text list "SINAMICS_G120_FW4.4_faults": 0 'No fault / Keine Störung'; 1000 'Internal software error / Softwarefehler intern'; 1001 'FloatingPoint exception / FloatingPoint Ausnahme'; 1002 'Internal software error / Softwarefehler intern'; 1003 'Acknowledgement delay when accessing the memory / Quittungsverzug bei Speicherzugriff'; 1004 'Internal software error / Softwarefehler intern'; 1005 'File upload/download error / Datei Upload/Download fehlgeschlagen'; 1009 'CU: Control module overtemperature / CU: Regelungsbaugruppe Übertemperatur'; 1010 'Drive type unknown / Antriebstyp unbekannt'; 1011 'Download interrupted / Download abgebrochen'; 1012 'Project conversion error / Projekt Konvertierungsfehler'; 1013 'CU: Fan operating time reached or exceeded / CU: Betriebsdauer Lüfter erreicht oder überschritten'; 1015 'Internal software error / Softwarefehler intern'; 1016 'Firmware changed / Firmware verändert'; 1017 'Component lists changed / Komponentenlisten verändert'; 1018 'Booting has been interrupted several times / Hochlauf mehrmals abgebrochen'; 1019 'Writing to the removable data medium unsuccessful / Wechselmedium schreiben fehlgeschlagen'; 1020 'Write to RAM disk unsuccessful / RAM disk schreiben fehlgeschlagen'; 1023 'Software timeout (internal) / Software Timeout intern'; 1028 'Configuration error / Konfigurationsfehler'; 1030 'Sign-of-life failure for master control / Lebenszeichenausfall bei Steuerungshoheit'; 1031 'Sign-of-life failure for OFF in REMOTE / Lebenszeichenausfall bei AUS in REMOTE'; 1033 'Units changeover: Reference parameter value invalid / Einheitenumschaltung: Bezugsparameterwert ungültig'; 1034 'Units changeover: Calculation parameter values after reference value change unsuccessful Einheitenumschaltung: Berechnung Parameterwerte nach Bezugswertänderung fehlgeschlagen'; 1035 'ACX: Boot from the back-up parameter back-up files / ACX: Hochlauf erfolgt aus Backup-Parametersicherungsdateien'; 1036 'ACX: Parameter back-up file missing / ACX: Parametersicherungsdatei fehlt'; 1037 'ACX: Re-naming the parameter back-up file unsuccessful / ACX: Parametersicherungsdatei umbenennen fehlgeschlagen'; 1038 'ACX: Loading the parameter back-up file unsuccessful / ACX: Parametersicherungsdatei laden fehlgeschlagen'; 1039 'ACX: Writing to the parameter back-up file was unsuccessful / ACX: Parametersicherungsdatei schreiben fehlgeschlagen'; 1040 'Save parameter settings and carry out a POWER ON / Parameter sichern und POWER ON erforderlich'; 1041 'Parameter save necessary / Parameter sichern erforderlich'; 1042 'Parameter error during project download / Parameterfehler beim Projekt-Download'; 1043 'Fatal error at project download / Schwerer Fehler beim Projekt-Download'; 1044 'CU: Descriptive data error / CU: Beschreibungsdaten fehlerhaft'; 1045 'CU: Configuring data invalid / CU: Projektierungsdaten ungültig'; 1049 'It is not possible to write to file / Schreiben in Datei nicht möglich'; 1050 'Memory card and device incompatible / Speicherkarte und Gerät inkompatibel'; 1053 'CU: System overload measured / CU: Systemüberlastung gemessen'; 1054 'CU: System limit exceeded / CU: Systemgrenze überschritten'; 1064 'CU: Internal error (CRC) / CU: Interner Fehler (CRC)'; 1066 'Buffer memory: 70% fill level reached or exceeded / Zwischenspeicher: Füllstand 70 % erreicht oder überschritten'; 1067 'Buffer memory: 100 % fill level reached / Zwischenspeicher: Füllstand 100 % erreicht'; 1068 'CU: Data memory, memory overflow / CU: Datenspeicher Speicherüberlauf'; 1069 'Parameter backup and device incompatible / Parametersicherung und Gerät inkompatibel'; 1098 'RTC: Date and time setting required / RTC: Datum und Zeit einstellen erforderlich'; 1099 'Tolerance window of time synchronization exited / Toleranzfenster der Uhrzeitsynchronisation verlassen'; 1100 'CU: Memory card withdrawn / CU: Speicherkarte gezogen'; 1104 'CU: Do not power down. File system being optimized. / CU: Nicht ausschalten Optimierung Dateisystem läuft'; 1105 'CU: Insufficient memory / CU: Speicher nicht ausreichend'; 1107 'CU: Data save in the non-volatile memory unsuccessful / CU: Speichern in nichtflüchtigen Speicher fehlgeschlagen'; 1110 'CU: More than one SINAMICS G on one Control Unit / CU: Mehr als ein SINAMICS G an einer Control Unit'; 1111 'CU: Mixed operation of drive units illegal / CU: Mischbetrieb von Antriebsgeräten unzulässig'; 1112 'CU: Power unit not permissible / CU: Leistungsteil unzulässig'; 1120 'Terminal initialization has failed / Initialisierung Klemmen fehlgeschlagen'; 1122 'Frequency at the measuring probe input too high / Frequenz am Messtastereingang zu hoch'; 1150 'CU: Number of instances of a drive object type exceeded / CU: Anzahl Instanzen eines Antriebsobjekttyps überschritten'; 1151 'CU: Number of drive objects of a category exceeded / CU: Anzahl Antriebsobjekte einer Kategorie überschritten'; 1200 'CU: Time slice management internal software error / CU: Zeitscheibenmanagement Softwarefehler intern'; 1205 'CU: Time slice overflow / CU: Zeitscheibenüberlauf'; 1221 'CU: Bas clk cyc too low / CU: Basistakt zu klein'; 1223 'CU: Sampling time inconsistent / CU: Abtastzeit inkonsistent'; 1224 'CU: Pulse frequency inconsistent / CU: Pulsfrequenz inkonsistent'; 1250 'CU: CU-EEPROM incorrect read-only data / CU: CU-EEPROM Read-Only-Daten fehlerhaft'; 1251 'CU: CU-EEPROM incorrect read-write data / CU: CU-EEPROM Read-Write-Daten fehlerhaft'; 1255 'CU: Option Board EEPROM read-only data error / CU: Option Board EEPROM Read-Only-Daten fehlerhaft'; 1256 'CU: Option Board EEPROM read-write data error / CU: Option Board EEPROM Read-Write-Daten fehlerhaft'; 1275 'Hardware description error / Hardware-Beschreibung fehlerhaft'; 1276 'Hardware description not fully compatible / Hardware-Beschreibung nicht voll kompatibel'; 1303 'Function not supported / Funktion nicht unterstützt'; 1305 'Topology: Component number missing / Topologie: Komponentennummer fehlt'; 1314 'Topology: Component must not be present / Topologie: Komponente darf nicht vorhanden sein'; 1315 'Drive object not ready for operation / Antriebsobjekt nicht betriebsfähig'; 1316 'Drive object inactive and again ready for operation / Antriebsobjekt inaktiv und wieder betriebsfähig'; 1317 'De-activated component again present / Deaktivierte Komponente wieder vorhanden'; 1318 'BICO: De-activated interconnections present / BICO: Aufgelöste Verschaltungen vorhanden'; 1319 'Inserted component not initialized / Zugesteckte Komponente nicht initialisiert'; 1320 'Topology: Drive object number does not exist in configuration / Topologie: Antriebsobjektnummer fehlt in Konfiguration'; 1321 'Topology: Drive object number does not exist in configuration Topologie: Antriebsobjektnummer existiert nicht in Konfiguration'; 1322 'Topology: Drive object number present twice in configuration Topologie: Antriebsobjektnummer zweimal in Konfiguration vorhanden'; 1323 'Topology: More than two partial lists created / Topologie: Mehr als zwei Teillisten angelegt'; 1324 'Topology: Dummy drive object number incorrectly created / Topologie: Dummy Antriebsobjektnummer falsch angelegt'; 1325 'Topology: Component Number not present in target topology Topologie: Komponentennummer nicht in Solltopologie enthalten'; 1330 'Topology: Quick commissioning not possible / Topologie: Schnellinbetriebnahme nicht möglich'; 1331 'Topology: At least one component not assigned to a drive object Topologie: Mindestens eine Komponente keinem Antriebsobjekt zugeordnet'; 1340 'Topology: Too many components on one line / Topologie: Zuviele Komponenten an einem Strang'; 1354 'Topology: Actual topology indicates an illegal component / Topologie: Isttopologie weist unzulässige Komponente auf'; 1355 'Topology: Actual topology changed / Topologie: Isttopologie geändert'; 1356 'Topology: Defective components in actual topology / Topologie: Defekte Komponente in Isttopologie'; 1360 'Topology: Actual topology not permissible / Topologie: Isttopologie unzulässig'; 1361 'Topology: Actual topology contains SINUMERIK and SIMOTION components Topologie: Isttopologie enthält SINUMERIK und SIMOTION Komponenten'; 1362 'Topology: Topology rule(s) broken / Topologie: Topologieregel nicht eingehalten'; 1375 'Topology: Actual topology, duplicate connection between two components Topologie: Isttopologie Verbindung doppelt zwischen zwei Komponenten'; 1380 'Topology: Actual topology, defective EEPROM / Topologie: Isttopologie defektes EEPROM'; 1381 'Topology: Comparison power unit shifted / Topologie: Vergleich Leistungsteil verschoben'; 1382 'Topology: Comparison Sensor Module shifted / Topologie: Vergleich Sensor Module verschoben'; 1383 'Topology: Comparison Terminal Module shifted / Topologie: Vergleich Terminal Module verschoben'; 1385 'Topology: Comparison CX32 shifted / Topologie: Vergleich CX32 verschoben'; 1387 'Topology: Comparison option slot component shifted / Topologie: Vergleich Option Slot Komponente verschoben'; 1388 'Topology: Comparison EnDat encoder shifted / Topologie: Vergleich EnDat-Geber verschoben'; 1416 'Topology: Comparison additional component in actual topology / Topologie: Vergleich Komponente zusätzlich in Isttopologie'; 1420 'Topology: Comparison a component is different / Topologie: Vergleich eine Komponente unterschiedlich'; 1425 'Topology: Comparison serial number of a component is different Topologie: Vergleich Seriennummer eine Komponente unterschiedlich'; 1428 'Topo: Comparison connection of a component is different Topologie: Vergleich Anschluss einer Komponente unterschiedlich'; 1429 'Topology: Comparison connection is different for more than one component Topologie: Vergleich Anschluss mehr als eine Komponente unterschiedlich'; 1451 'Topology: Target topology is invalid / Topologie: Solltopologie ungültig'; 1470 'Topology:Target topology ring-type connection detected / Topologie: Solltopologie Ringverbindung erkannt'; 1475 'Topology: Target topology duplicate connection between two components Topologie: Solltopologie Verbindung doppelt zwischen zwei Komponenten'; 1481 'Topology: Comparison power unit missing in the actual topology Topologie: Vergleich Leistungsteil in Isttopologie fehlt'; 1482 'Topology: Comparison Sensor Module missing in the actual topology Topologie: Vergleich Sensor Module in Isttopologie fehlt'; 1483 'Topology: Comparison Terminal Module missing in the actual topology Topologie: Vergleich Terminal Module in Isttopologie fehlt'; 1485 'Topology: Comparison CX32 missing in the actual topology / Topologie: Vergleich CX32 in Isttopologie fehlt'; 1487 'Topology: Comparison option slot components missing in the actual topology Topologie: Vergleich Option Slot Komponente in Isttopologie fehlt'; 1488 'Topology: Comparison EnDat encoder missing in the actual topology Topologie: Vergleich EnDat-Geber in Isttopologie fehlt'; 1505 'BICO: Interconnection cannot be established / BICO: Verschaltung kann nicht hergestellt werden'; 1506 'BICO: No standard telegram / BICO: Kein Standardtelegramm'; 1507 'BICO: Interconnections to inactive objects present / BICO: Verschaltungen zu inaktiven Objekten vorhanden'; 1508 'BICO: Interconnections to inactive objects exceeded / BICO: Verschaltungen zu inaktiven Objekten überschritten'; 1510 'BICO: Signal source is not float type / BICO: Signalquelle ist nicht Float'; 1511 'BICO: Interconnection with different scalings / BICO: Verschaltung mit unterschiedlicher Normierung'; 1512 'BICO: No scaling available / BICO: Keine Normierung vorhanden'; 1513 'BICO: Interconnection cross DO with different scalings BICO: Verschaltung DO-übergreifend mit unterschiedlicher Normierung'; 1514 'BICO: Error when writing during a reconnect / BICO: Fehler beim Schreiben während Reconnect'; 1515 'BICO: Writing to parameter not permitted as the master control is active BICO: Parameterschreiben nicht erlaubt da Steuerungshoheit aktiv'; 1590 'Drive: Motor maintenance interval expired / Antrieb: Motor Wartungsintervall abgelaufen'; 1600 'SI CU: STOP A initiated / SI CU: STOP A ausgelöst'; 1611 'SI CU: Defect in a monitoring channel / SI CU: Defekt in einem Überwachungskanal'; 1612 'SI CU: STO inputs for power units connected in parallel different SI CU: STO-Eingänge bei parallelgeschalteten Leistungsteilen unterschiedlich'; 1620 'SI CU: Safe Torque Off active / SI CU: Sicher abgeschaltetes Moment aktiv'; 1621 'SI CU: Safe Stop 1 active / SI CU: Safe Stop 1 aktiv'; 1625 'SI CU: Sign-of-life error in safety data / SI CU: Lebenszeichen in Safety-Daten fehlerhaft'; 1630 'SI CU: Brake control error / SI CU: Bremsenansteuerung fehlerhaft'; 1649 'SI CU: Internal software error / SI CU: Softwarefehler intern'; 1650 'SI CU: Acceptance test required / SI CU: Abnahmetest erforderlich'; 1651 'SI CU: Synchronization safety time slices unsuccessful / SI CU: Synchronisation Safety-Zeitscheiben fehlgeschlagen'; 1652 'SI CU: Illegal monitoring clock cycle / SI CU: Überwachungstakt unzulässig'; 1653 'SI CU: PROFIBUS configuration error / SI CU: PROFIBUS-Projektierung fehlerhaft'; 1655 'SI CU: Align monitoring functions / SI CU: Abgleich der Überwachungsfunktionen'; 1656 'SI CU: Motor Module parameter error / SI CU: Parameter Motor Module fehlerhaft'; 1659 'SI CU: Write request for parameter rejected / SI CU: Schreibauftrag für Parameter abgewiesen'; 1660 'SI CU: Safety-related functions not supported / SI CU: Sichere Funktionen nicht unterstützt'; 1662 'Error internal communications / Fehler interne Kommunikation'; 1663 'SI CU: Copying the SI parameters rejected / SI CU: Kopieren der SI-Parameter abgelehnt'; 1664 'SI CU: No automatic firmware update / SI CU: Kein automatischer Firmware-Update'; 1665 'SI CU: System is defective / SI CU: System ist defekt'; 1666 'SI Motion CU: Steady-state (static) 1 signal at the F-DI for safety-relevant acknowledgement SI Motion CU: Statisches 1-Signal am F-DI für sichere Quittierung'; 1669 'SI Motion: Unfavorable combination of motor and power unit SI Motion: Kombination von Motor und Leistungsteil ungünstig'; 1670 'SI Motion: Invalid parameterization Sensor Module / SI Motion: Parametrierung Sensor Module ungültig'; 1671 'SI Motion: Parameterization encoder error / SI Motion: Parametrierung Geber fehlerhaft'; 1672 'SI CU: Motor Module software/hardware incompatible / SI CU: Motor Module Software/Hardware inkompatibel'; 1673 'SI Motion: Sensor Module software/hardware incompatible / SI Motion: Sensor Module Software/Hardware inkompatibel'; 1680 'SI Motion CU: Checksum error safety monitoring functions / SI Motion CU: Prüfsummenfehler sichere Überwachungen'; 1681 'SI Motion CU: Incorrect parameter value / SI Motion CU: Parameterwert falsch'; 1682 'SI Motion CU: Monitoring function not supported / SI Motion CU: Überwachungsfunktion nicht unterstützt'; 1683 'SI Motion CU: SOS/SLS enable missing / SI Motion CU: SOS/SLS-Freigabe fehlt'; 1684 'SI Motion: Safely limited position limit values interchanged / SI Motion: Sicher begrenzte Position Grenzwerte vertauscht'; 1685 'SI Motion CU: Safely-limited speed limit value too high SI Motion CU: Sicher begrenzte Geschwindigkeit Grenzwert zu groß'; 1686 'SI Motion: Illegal parameterization cam position / SI Motion: Parametrierung Nockenposition unzulässig'; 1687 'SI Motion: Illegal parameterization modulo value SCA (SN) / SI Motion: Parametrierung Modulowert SCA (SN) unzulässig'; 1688 'SI Motion CU: Actual value synchronization not permissible / SI Motion CU: Istwertsynchronisation nicht zulässig'; 1689 'SI Motion: Axis re-configured / SI Motion: Achse umkonfiguriert'; 1690 'SI Motion: Data save problem for the NVRAM / SI Motion: Datensicherungsproblem beim NVRAM'; 1691 'SI Motion: Ti and To unsuitable for DP cycle / SI Motion: Ti und To ungeeignet für den DP-Takt'; 1692 'SI Motion CU: Parameter value not permitted for encoderless / SI Motion CU: Parameterwert geberlos unzulässig'; 1693 'SI CU: Safety parameter settings changed, warm restart/POWER ON required SI CU: Safety-Parametrierung geändert Warmstart/POWER ON erforderlich'; 1694 'SI Motion CU: Firmware version Motor Module older Control Unit SI Motion CU: Firmware-Version Motor Module älter Control Unit'; 1695 'SI Motion: Sensor Module was replaced / SI Motion: Sensor Module wurde getauscht'; 1696 'SI Motion: Testing of the motion monitoring functions selected when booting SI Motion: Testanwahl der Bewegungsüberwachungen im Hochlauf'; 1697 'SI Motion: Motion monitoring functions must be tested / SI Motion: Test der Bewegungsüberwachungen erforderlich'; 1698 'SI CU: Commissioning mode active / SI CU: Inbetriebnahmemodus aktiv'; 1699 'SI CU: Shutdown path must be tested / SI CU: Test der Abschaltpfade erforderlich'; 1700 'SI Motion CU: STOP A initiated / SI Motion CU: STOP A ausgelöst'; 1701 'SI Motion CU: STOP B initiated / SI Motion CU: STOP B ausgelöst'; 1706 'SI Motion CU: SAM/SBR limit exceeded / SI Motion CU: SAM/SBR Grenze überschritten'; 1707 'SI Motion CU: Tolerance for safe operating stop exceeded / SI Motion CU: Toleranz für Sicheren Betriebshalt überschritten'; 1708 'SI Motion CU: STOP C initiated / SI Motion CU: STOP C ausgelöst'; 1709 'SI Motion CU: STOP D initiated / SI Motion CU: STOP D ausgelöst'; 1710 'SI Motion CU: STOP E initiated / SI Motion CU: STOP E ausgelöst'; 1711 'SI Motion CU: Defect in a monitoring channel / SI Motion CU: Defekt in einem Überwachungskanal'; 1712 'SI Motion CU: Defect in F-IO processing / SI Motion CU: Defekt bei F-IO-Verarbeitung'; 1714 'SI Motion CU: Safely-Limited Speed exceeded / SI Motion CU: Sicher begrenzte Geschwindigkeit überschritten'; 1715 'SI Motion CU: Safely-Limited Position exceeded / SI Motion CU: Sicher begrenzte Position überschritten'; 1716 'SI Motion CU: Tolerance for safe motion direction exceeded SI Motion CU: Toleranz für sichere Bewegungsrichtung überschritten'; 1745 'SI Motion CU: Checking braking torque for the brake test / SI Motion CU: Bremsmoment beim Bremsentest überprüfen'; 1750 'SI Motion CU: Hardware fault safety-relevant encoder / SI Motion CU: Hardware-Fehler sicherer Geber'; 1751 'SI Motion CU: Effectivity test error safety-relevant encoder / SI Motion CU: Wirksamkeitstest-Fehler sicherer Geber'; 1770 'SI Motion CU: Discrepancy error of the failsafe inputs or outputs SI Motion CU: Diskrepanzfehler der fehlersicheren Eingänge oder Ausgänge'; 1772 'SI Motion CU: Test stop failsafe inputs/outputs active / SI Motion CU: Teststop fehlersichere Eingänge/Ausgänge aktiv'; 1773 'SI Motion CU: Test stop error / SI Motion CU: Teststop fehlerhaft'; 1774 'SI Motion CU: Test stop necessary / SI Motion CU: Teststop notwendig'; 1796 'SI Motion CU: Wait for communication / SI Motion CU: Warten auf Kommunikation'; 1797 'SI Motion CU: Axis not safely referenced / SI Motion CU: Achse nicht sicher referenziert'; 1798 'SI Motion CU: Test stop running / SI Motion CU: Teststop läuft'; 1799 'SI Motion CU: Acceptance test mode active / SI Motion CU: Abnahmetestmodus aktiv'; 1840 'SMI: Component found without motor data / SMI: Komponente ohne Motordaten gefunden'; 1900 'PB/PN: Configuration telegram error / PB/PN: Konfigurationstelegramm fehlerhaft'; 1902 'IF1: PB/PN clock cycle synchronous operation parameterization not permissible IF1: PB/PN Taktsynchroner Betrieb Parametrierung unzulässig'; 1903 'COMM INT: Receive configuration data invalid / COMM INT: Empfangs-Konfigurationsdaten ungültig'; 1910 'Fieldbus interface setpoint timeout / Feldbus SS Sollwert Timeout'; 1911 'PB/PN clock cycle synchronous operation clock cycle failure / PB/PN Taktsynchroner Betrieb Taktausfall'; 1912 'PB/PN clock cycle synchronous operation sign-of-life failure / PB/PN Taktsynchroner Betrieb Lebenszeichenausfall'; 1913 'COMM INT: Monitoring time sign-of-life expired / COMM INT: Überwachungszeit Lebenszeichen abgelaufen'; 1914 'COMM INT: Monitoring time configuration expired / COMM INT: Überwachungszeit Konfiguration abgelaufen'; 1915 'PB/PN clock cycle synchronous operation sign-of-life failure drive object 1 PB/PN Taktsynchroner Betrieb Lebenszeichenausfall Antriebsobjekt 1'; 1920 'PROFIBUS: Interruption cyclic connection / PROFIBUS: Unterbrechung zyklische Verbindung'; 1921 'PROFIBUS: Receive setpoints after To / PROFIBUS: Sollwerte nach To empfangen'; 1930 'PB/PN current controller clock cycle clock cycle synch. not equal PB/PN Stromreglertakt taktsynchron ungleich'; 1931 'PB/PN speed controller clock cycle clock cycle synch. not equal / PB/PN Drehzahlreglertakt taktsynchron ungleich'; 1932 'PB/PN clock cycle synchronization missing for DSC / PB/PN Taktsynchronisation fehlt bei DSC'; 1940 'PB/PN clock cycle synchronism not reached / PB/PN Taktsynchronität nicht erreicht'; 1941 'PB/PN clock cycle signal missing when establishing bus communication PB/PN Taktsignal fehlt beim Busaufbau'; 1943 'PB/PN clock cycle signal error when establishing bus communication PB/PN Taktsignal beim Busaufbau gestört'; 1944 'PB/PN sign-of-life synchronism not reached / PB/PN Lebenszeichensynchronität nicht erreicht'; 1945 'PROFIBUS: Connection to the Publisher failed / PROFIBUS: Verbindung zum Publisher gestört'; 1946 'PROFIBUS: Connection to the Publisher aborted / PROFIBUS: Verbindung zum Publisher abgebrochen'; 1950 'PB/PN clock cycle synchronous operation synchronization unsuccessful PB/PN Taktsynchroner Betrieb Synchronisation fehlgeschlagen'; 1951 'CU SYNC: Synchronization application clock cycle missing / CU SYNC: Synchronisation Applikationstakt fehlt'; 1953 'CU SYNC: Synchronization not completed / CU SYNC: Synchronisation nicht abgeschlossen'; 1980 'PN: Interruption cyclic connection / PN: Unterbrechung zyklische Verbindung'; 1981 'PN: Maximum number of controllers exceeded / PN: Maximale Anzahl Controller überschritten'; 1982 'PROFINET: Second controller missing / PROFINET: Zweiter Controller fehlt'; 1989 'PROFINET: Internal cyclic data transfer error / PROFINET: Interner Fehler bei zyklischer Datenübertragung'; 1990 'USS: PZD configuration error / USS: PZD Konfiguration fehlerhaft'; 2000 'Function generator: Start not possible / Funktionsgenerator: Start nicht möglich'; 2005 'Function generator: Drive does not exist / Funktionsgenerator: Antrieb existiert nicht'; 2006 'Function generator: No drive specified for connection / Funktionsgenerator: Kein Antrieb zur Aufschaltung angegeben'; 2007 'Function generator: Drive not SERVO / VECTOR / DC_CTRL / Funktionsgenerator: Antrieb kein SERVO/VECTOR/DC_CTRL'; 2008 'Function generator: Drive specified a multiple number of times / Funktionsgenerator: Antrieb mehrfach angegeben'; 2009 'Function generator: Illegal mode / Funktionsgenerator: Betriebsart unzulässig'; 2010 'Function generator: Speed setpoint from the drive is not zero / Funktionsgenerator: Drehzahlsollwert von Antrieb nicht Null'; 2011 'Function generator: The actual drive speed is not zero / Funktionsgenerator: Drehzahlistwert von Antrieb nicht Null'; 2015 'Function generator: Drive enable signals missing / Funktionsgenerator: Antriebsfreigaben fehlen'; 2016 'Function generator: Magnetizing running / Funktionsgenerator: Aufmagnetisierung läuft'; 2020 'Function generator: Parameter cannot be changed / Funktionsgenerator: Parameter nicht änderbar'; 2025 'Function generator: Period too short / Funktionsgenerator: Periodendauer zu klein'; 2026 'Function generator: Pulse width too high / Funktionsgenerator: Pulsbreite zu groß'; 2030 'Function generator: Physical address equals zero / Funktionsgenerator: Physikalische Adresse gleich Null'; 2040 'Function generator: Illegal value for offset / Funktionsgenerator: Wert für Offset unzulässig'; 2041 'Function generator: Illegal value for bandwidth / Funktionsgenerator: Wert für Bandbreite unzulässig'; 2047 'Function generator: Time slice clock cycle invalid / Funktionsgenerator: Zeitscheibentakt ungültig'; 2050 'Trace: Start not possible / Trace: Start nicht möglich'; 2055 'Trace: Recording time too short / Trace: Aufzeichnungsdauer zu klein'; 2056 'Trace: Recording cycle too short / Trace: Aufzeichnungstakt zu klein'; 2057 'Trace: Time slice clock cycle invalid / Trace: Zeitscheibentakt ungültig'; 2058 'Trace: Time slice clock cycle for endless trace not valid / Trace: Zeitscheibentakt für Endlostrace ungültig'; 2059 'Trace: Time slice clock cycle for 2 x 8 recording channels not valid Trace: Zeitscheibentakt für 2 x 8 Aufzeichnungskanäle ungültig'; 2060 'Trace: Signal to be traced missing / Trace: Aufzuzeichnendes Signal fehlt'; 2061 'Trace: Invalid signal / Trace: Signal ungültig'; 2062 'Trace: Invalid trigger signal / Trace: Triggersignal ungültig'; 2063 'Trace: Invalid data type / Trace: Datentyp ungültig'; 2070 'Trace: Parameter cannot be changed / Trace: Parameter nicht änderbar'; 2075 'Trace: Pretrigger time too long / Trace: Pretriggerzeit zu groß'; 2080 'Trace: Parameterization deleted due to unit changeover / Trace: Parametrierung wegen Einheitenumschaltung gelöscht'; 2099 'Trace: Insufficient Control Unit memory / Trace: Speicherplatz der Control Unit nicht ausreichend'; 2100 'Drive: Computing dead time current controller too short / Antrieb: Rechentotzeit Stromregler zu klein'; 2150 'OA: Application cannot be loaded / OA: Applikation nicht ladbar'; 2151 'OA: Internal software error / OA: Softwarefehler intern'; 2152 'OA: Insufficient memory / OA: Speicher nicht ausreichend'; 3000 'NVRAM fault on action / NVRAM Fehler bei Aktion'; 3001 'NVRAM checksum incorrect / NVRAM Prüfsumme fehlerhaft'; 3500 'TM: Initialization / TM: Initialisierung'; 3501 'TM: Sampling time change / TM: Abtastzeiten Änderung'; 3505 'CU: Analog input wire breakage / CU: Analogeingang Drahtbruch'; 3506 '24 V power supply missing / Spannungsversorgung 24 V fehlt'; 3507 'Digital output not set / Digitalausgang nicht gesetzt'; 3510 'CU: Calibration data not plausible / CU: Kalibrierdaten nicht plausibel'; 3520 'CU: Temperature sensor fault / CU: Fehler Temperatursensor'; 3550 'TM: Speed setpoint filter natural frequency > Shannon frequency TM: Drehzahlsollwertfilter Eigenfrequenz > Shannon-Frequenz'; 3590 'TM: Module not ready / TM: Modul nicht bereit'; 5000 'Power unit: Overtemperature heat sink AC inverter / Leistungsteil: Übertemperatur Kühlkörper Wechselrichter'; 5001 'Power unit: Overtemperature depletion layer chip / Leistungsteil: Übertemperatur Sperrschicht Chip'; 5002 'Power unit: Air intake overtemperature / Leistungsteil: Übertemperatur Zuluft'; 5003 'Power unit: Internal overtemperature / Leistungsteil: Übertemperatur Innenraum'; 5004 'Power unit: Rectifier overtemperature / Leistungsteil: Übertemperatur Gleichrichter'; 5005 'Cooling system: Cooling medium flow rate too low / Rückkühlanlage: Kühlmittel Volumenstrom zu klein'; 5006 'Power unit: Overtemperature thermal model / Leistungsteil: Übertemperatur Thermisches Modell'; 5007 'Power unit: Overtemperature thermal model (chassis PU) / Leistungsteil: Übertemperatur Thermisches Modell (Chassis-LT)'; 5054 'Parallel circuit: Power unit de-activated / Parallelschaltung: Leistungsteil deaktiviert'; 5055 'Parallel connection: Power units with illegal code numbers Parallelschaltung: Leistungsteile mit unzulässigen Codenummern'; 5056 'Parallel circuit: Power unit EPROM versions differ Parallelschaltung: Leistungsteil EPROM-Versionen unterschiedlich'; 5057 'Parallel circuit: Power unit firmware versions differ Parallelschaltung: Leistungsteil Firmware-Versionen unterschiedlich'; 5058 'Parallel circuit: VSM EEPROM versions differ / Parallelschaltung: VSM EEPROM-Versionen unterschiedlich'; 5059 'Parallel circuit: VSM firmware versions differ / Parallelschaltung: VSM Firmware-Versionen unterschiedlich'; 5060 'Parallel circuit: Power unit firmware version does not match / Parallelschaltung: Leistungsteil Firmware-Version nicht passend'; 5061 'Infeed, number of VSM / Einspeisung VSM Anzahl'; 6310 'Supply voltage (p0210) incorrectly parameterized / Anschlussspannung (p0210) fehlerhaft parametriert'; 6921 'Braking resistor phase unsymmetry / Bremswiderstand Phasenunsymmetrie'; 6922 'Braking resistor phase failure / Bremswiderstand Phasenausfall'; 7011 'Drive: Motor overtemperature / Antrieb: Motor Übertemperatur'; 7012 'Drive: I2t motor model overtemperature / Antrieb: I2t Motormodell Übertemperatur'; 7015 'Drive: Motor temperature sensor alarm / Antrieb: Motortemperatursensor Warnung'; 7016 'Drive: Motor temperature sensor fault / Antrieb: Motortemperatursensor Störung'; 7042 'Drive: Motor data identification routine completed / Antrieb: Motordatenidentifikation beendet'; 7043 'Drive: Speed controller optimization completed / Antrieb: Drehzahlregleroptimierung beendet'; 7044 'Drive: Pole position identification completed / Antrieb: Pollageidentifikation beendet'; 7045 'Drive: Friction characteristic record completed / Antrieb: Reibkennlinie Record beendet'; 7080 'Drive: Incorrect control parameter / Antrieb: Regelungsparameter fehlerhaft'; 7082 'Macro: Execution not possible / Makro: Ausführung nicht möglich'; 7083 'Macro: ACX file not found / Makro: ACX-File nicht gefunden'; 7084 'Macro: Condition for WaitUntil not fulfilled / Makro: Bedingung für WaitUntil nicht erfüllt'; 7085 'Drive: Open-loop/closed-loop control parameters changed / Antrieb: Parameter der Steuerung/Regelung geändert'; 7086 'Units changeover: Parameter limit violation due to reference value change Einheitenumschaltung: Parametergrenzverletzung durch Bezugswertänderung'; 7087 'Drive: Encoderless operation not possible for the selected pulse frequency Antrieb: Geberloser Betrieb bei eingestellter Pulsfrequenz nicht möglich'; 7088 'Units changeover: Parameter limit violation due to units changeover Einheitenumschaltung: Parametergrenzverletzung durch Einheitenumschaltung'; 7089 'Changing over units: Function module activation is blocked because the units have been changed over Einheitenumschaltung: Funktionsmodul aktivieren ist blockiert weil Einheiten umgeschaltet wurden'; 7090 'Drive: Upper torque limit less than the lower torque limit / Antrieb: Drehmomentgrenze oben kleiner unten'; 7100 'Drive: Sampling times cannot be reset / Antrieb: Abtastzeiten nicht zurücksetzbar'; 7110 'Drive: Sampling times and basic clock cycle do not match / Antrieb: Abtastzeiten und Basistakt nicht passend'; 7200 'Drive: Master control ON command present / Antrieb: Steuerungshoheit EIN-Befehl steht an'; 7220 'Drive: Master control by PLC missing / Antrieb: Führung durch PLC fehlt'; 7300 'Drive: Line contactor feedback signal missing / Antrieb: Netzschütz Rückmeldung fehlt'; 7311 'Bypass motor switch / Bypass Motorschalter'; 7312 'Bypass LSS: / Bypass Netzschalter'; 7320 'Drive: Automatic restart interrupted / Antrieb: Automatischer Wiederanlauf abgebrochen'; 7321 'Drive: Automatic restart active / Antrieb: Automatischer Wiederanlauf aktiv'; 7324 'Drive: Hibernation active - drive powers itself down / Antrieb: Hibernation aktiv - Antrieb schaltet sich aus'; 7325 'Drive: Hibernation active - drive re-activated automatically Antrieb: Hibernation aktiv - Antrieb schaltet automatisch wieder ein'; 7329 'Drive: kT estimator, kT(iq) characteristic or voltage compensation does not function Antrieb: kT-Schätzer, kT(iq)-Kennlinie oder Spannungskompensation nicht funktionsfähig'; 7330 'Flying restart: Measured search current too low / Fangen: Gemessener Suchstrom zu klein'; 7331 'Flying restart: Function not supported / Fangen: Funktion nicht unterstützt'; 7350 'Drive: Measuring probe parameterized to a digital output / Antrieb: Messtaster auf Digitalausgang parametriert'; 7400 'Drive: DC link voltage maximum controller active / Antrieb: Zwischenkreisspannungs-Maximum-Regler aktiv'; 7401 'Drive: DC link voltage maximum controller de-activated / Antrieb: Zwischenkreisspannungs-Maximum-Regler deaktiviert'; 7402 'Drive: DC link voltage minimum controller active / Antrieb: Zwischenkreisspannungs-Minimum-Regler aktiv'; 7403 'Drive: Lower DC link voltage threshold reached / Antrieb: Zwischenkreisspannungsschwelle unten erreicht'; 7404 'Drive: Upper DC link voltage threshold reached / Antrieb: Zwischenkreisspannungsschwelle oben erreicht'; 7405 'Drive: Kinetic buffering minimum speed not reached / Antrieb: Kinetische Pufferung minimale Drehzahl unterschritten'; 7406 'Drive: Kinetic buffering maximum time exceeded / Antrieb: Kinetische Pufferung maximale Dauer überschritten'; 7409 'Drive: U/f control, current limiting controller active / Antrieb: U/f-Steuerung Strombegrenzungsregler aktiv'; 7410 'Drive: Current controller output limited / Antrieb: Stromreglerausgang begrenzt'; 7411 'Drive: Flux controller output limited / Antrieb: Flussreglerausgang begrenzt'; 7412 'Drive: Commutation angle incorrect (motor model) / Antrieb: Kommutierungswinkel fehlerhaft (Motormodell)'; 7413 'Drive: Commutation angle incorrect (pole position identification) / Antrieb: Kommutierungswinkel fehlerhaft (Pollageidentifikation)'; 7414 'Drive: Encoder serial number changed / Antrieb: Geberseriennummer geändert'; 7415 'Drive: Angular commutation offset transfer running / Antrieb: Übertragung Kommutierungswinkeloffset läuft'; 7416 'Drive: Flux controller configuration / Antrieb: Konfiguration Flussregler'; 7417 'Drive: Pulse technique not plausible (motor model) / Antrieb: Pulsverfahren nicht plausibel (Motormodell)'; 7418 'Drive: Higher current controller dynamic performance possible / Antrieb: Höhere Stromreglerdynamik möglich'; 7420 'Drive: Current setpoint filter natural frequency > Shannon frequency Antrieb: Stromsollwertfilter Eigenfrequenz > Shannon-Frequenz'; 7421 'Drive: Speed filter natural frequency > Shannon frequency / Antrieb: Drehzahlfilter Eigenfrequenz > Shannon-Frequenz'; 7422 'Drive: Reference model natural frequency > Shannon frequency Antrieb: Referenzmodell Eigenfrequenz > Shannon-Frequenz'; 7426 'Technology controller actual value limited / Technologieregler Istwert begrenzt'; 7427 'Motor staging alarm / Motor Staging Warnung'; 7429 'Drive: DSC without encoder not possible / Antrieb: DSC ohne Geber nicht möglich'; 7430 'Drive: Changeover to open-loop torque controlled operation not possible Antrieb: Umschaltung Drehmomentgesteuerter Betrieb nicht möglich'; 7431 'Drive: Changeover to encoderless operation not possible / Antrieb: Umschaltung Geberloser Betrieb nicht möglich'; 7432 'Drive: Motor without overvoltage protection / Antrieb: Motor ohne Überspannungsschutz'; 7433 'Drive: Closed-loop control with encoder is not possible as the encoder has not been unparked Antrieb: Regelung mit Geber nicht möglich da Geber nicht entparkt'; 7434 'Drive: It is not possible to change the direction of rotation with the pulses enabled Antrieb: Drehsinn ändern unter Impulsfreigabe nicht möglich'; 7435 'Drive: Setting the ramp-function generator for sensorless vector control Antrieb: Hochlaufgebersetzen bei geberloser Vektorregelung'; 7436 'Free tec_ctrl 0 actual value limited / Freier Tec_reg 0 Istwert begrenzt'; 7437 'Free tec_ctrl 1 actual value limited / Freier Tec_reg 1 Istwert begrenzt'; 7438 'Free tec_ctrl 2 actual value limited / Freier Tec_reg 2 Istwert begrenzt'; 7439 'Drive: Higher current controller dynamic performance not possible Antrieb: Höhere Stromreglerdynamik nicht möglich'; 7440 'EPOS: Jerk time is limited / EPOS: Ruckzeit wird begrenzt'; 7441 'LR: Save the position offset of the absolute encoder adjustment LR: Lageoffset der Absolutwertgeberjustage sichern'; 7442 'LR: Multiturn does not match the modulo range / LR: Multiturn passt nicht zum Modulobereich'; 7443 'LR: Reference point coordinate not in the permissible range / LR: Referenzpunkt-Koordinate nicht im zulässigen Bereich'; 7446 'Load gear: Position tracking cannot be reset / Lastgetriebe: Lageverfolgung lässt sich nicht zurücksetzen'; 7447 'Load gear: Position tracking, maximum actual value exceeded / Lastgetriebe: Lageverfolgung maximaler Istwert überschritten'; 7448 'Load gear: Position tracking, linear axis has exceeded the maximum range Lastgetriebe: Lageverfolgung Linearachse hat maximalen Bereich überschritten'; 7449 'Load gear: Position tracking, actual position outside tolerance window Lastgetriebe: Lageverfolgung Aktuelle Position außerhalb Toleranzfenster'; 7450 'LR: Standstill monitoring has responded / LR: Stillstandsüberwachung hat angesprochen'; 7451 'LR: Position monitoring has responded / LR: Positionierüberwachung hat angesprochen'; 7452 'LR: Following error too high / LR: Schleppabstand zu groß'; 7453 'LR: Position actual value preprocessing error / LR: Lageistwertaufbereitung fehlerhaft'; 7454 'LR: Position actual value preprocessing does not have a valid encoder LR: Lageistwertaufbereitung hat keinen gültigen Geber'; 7455 'EPOS: Maximum velocity limited / EPOS: Maximalgeschwindigkeit begrenzt'; 7456 'EPOS: Setpoint velocity limited / EPOS: Sollgeschwindigkeit begrenzt'; 7457 'EPOS: Combination of input signals illegal / EPOS: Eingangssignale Kombination unzulässig'; 7458 'EPOS: Reference cam not found / EPOS: Referenznocken nicht gefunden'; 7459 'EPOS: No zero mark / EPOS: Keine Nullmarke vorhanden'; 7460 'EPOS: End of reference cam not found / EPOS: Referenznockenende nicht gefunden'; 7461 'EPOS: Reference point not set / EPOS: Referenzpunkt nicht gesetzt'; 7462 'EPOS: Selected traversing block number does not exist / EPOS: Angewählte Verfahrsatznummer existiert nicht'; 7463 'EPOS: External block change not requested in the traversing block EPOS: Externer Satzwechsel im Verfahrsatz nicht angefordert'; 7464 'EPOS: Traversing block is inconsistent / EPOS: Verfahrsatz ist inkonsistent'; 7465 'EPOS: Traversing block does not have a subsequent block / EPOS: Verfahrsatz hat keinen Folgesatz'; 7466 'EPOS: Traversing block number assigned a multiple number of times EPOS: Verfahrsatznummer mehrfach vergeben'; 7467 'EPOS: Traversing block has illegal task parameters / EPOS: Verfahrsatz hat unzulässigen Auftragsparameter'; 7468 'EPOS: Traversing block jump destination does not exist / EPOS: Verfahrsatz Sprungziel existiert nicht'; 7469 'EPOS: Traversing block < target position < software limit switch minus EPOS: Verfahrsatz Zielposition < Software-Endschalter Minus'; 7470 'EPOS: Traversing block> target position > software limit switch plus EPOS: Verfahrsatz Zielposition > Software-Endschalter Plus'; 7471 'EPOS: Traversing block target position outside the modulo range EPOS: Verfahrsatz Zielposition außerhalb Modulobereich'; 7472 'EPOS: Traversing block ABS_POS/ABS_NEG not possible / EPOS: Verfahrsatz ABS_POS/ABS_NEG nicht möglich'; 7473 'EPOS: Beginning of traversing range reached / EPOS: Verfahrbereichsanfang angefahren'; 7474 'EPOS: End of traversing range reached / EPOS: Verfahrbereichsende angefahren'; 7475 'EPOS: Target position < start of traversing range / EPOS: Zielposition < Verfahrbereichsanfang'; 7476 'EPOS: Target position > end of the traversing range / EPOS: Zielposition > Verfahrbereichsende'; 7477 'EPOS: Target position < software limit switch minus / EPOS: Zielposition < Software-Endschalter Minus'; 7478 'EPOS: Target position > software limit switch plus / EPOS: Zielposition > Software-Endschalter Plus'; 7479 'EPOS: Software limit switch minus reached / EPOS: Software-Endschalter Minus angefahren'; 7480 'EPOS: Software limit switch plus reached / EPOS: Software-Endschalter Plus angefahren'; 7481 'EPOS: Axis position < software limit switch minus / EPOS: Achsposition < Software-Endschalter Minus'; 7482 'EPOS: Axis position > software limit switch plus / EPOS: Achsposition > Software-Endschalter Plus'; 7483 'EPOS: Travel to fixed stop clamping torque not reached / EPOS: Fahren auf Festanschlag Klemmmoment nicht erreicht'; 7484 'EPOS: Fixed stop outside the monitoring window / EPOS: Festanschlag außerhalb Überwachungsfenster'; 7485 'EPOS: Fixed stop not reached / EPOS: Festanschlag nicht erreicht'; 7486 'EPOS: Intermediate stop missing / EPOS: Zwischenhalt fehlt'; 7487 'EPOS: Reject traversing task missing / EPOS: Verfahrauftrag verwerfen fehlt'; 7488 'EPOS: Relative positioning not possible / EPOS: Relative Positionierung nicht möglich'; 7489 'EPOS: Reference point correction outside the window / EPOS: Referenzpunktkorrektur außerhalb Fenster'; 7490 'EPOS: Enable signal withdrawn while traversing / EPOS: Freigabe während Verfahren weggenommen'; 7491 'EPOS: STOP cam minus reached / EPOS: STOP-Nocken Minus angefahren'; 7492 'EPOS: STOP cam plus reached / EPOS: STOP-Nocken Plus angefahren'; 7493 'LR: Overflow of the value range for position actual value / LR: Überlauf des Wertebereiches für Lageistwert'; 7494 'LR: Drive Data Set changeover in operation / LR: Antriebsdatensatz-Umschaltung während Betrieb'; 7495 'LR: Reference function interrupted / LR: Referenzfunktion abgebrochen'; 7496 'EPOS: Enable not possible / EPOS: Freigabe nicht möglich'; 7497 'LR: Position setting value activated / LR: Lagesetzwert aktiviert'; 7498 'LR: Measuring probe evaluation not possible / LR: Messtasterauswertung nicht möglich'; 7499 'EPOS: Reversing cam approached with the incorrect traversing direction EPOS: Umkehrnocken mit falscher Verfahrrichtung angefahren'; 7500 'Drive: Power unit data set PDS not configured / Antrieb: Leistungsteildatensatz PDS nicht projektiert'; 7501 'Drive: Motor Data Set MDS not configured / Antrieb: Motordatensatz MDS nicht projektiert'; 7502 'Drive: Encoder Data Set EDS not configured / Antrieb: Geberdatensatz EDS nicht projektiert'; 7503 'EPOS: STOP cam approached with the incorrect traversing direction EPOS: STOP-Nocken mit falscher Verfahrrichtung angefahren'; 7504 'Drive: Motor data set is not assigned to a drive data set Antrieb: Motordatensatz ist keinem Antriebsdatensatz zugeordnet'; 7505 'EPOS: Travel to fixed stop not possible in the V/f control mode EPOS: Fahren auf Festanschlag im U/f-Steuerungs-Betrieb nicht möglich'; 7509 'Drive: Component number missing / Antrieb: Komponentennummer fehlt'; 7510 'Drive: Identical encoder in the drive data set / Antrieb: Identische Geber im Antriebsdatensatz'; 7511 'Drive: Encoder used a multiple number of times / Antrieb: Geber mehrfach verwendet'; 7512 'Drive: Encoder data set changeover cannot be parameterized / Antrieb: Geberdatensatzumschaltung nicht parametrierbar'; 7514 'Drive: Data structure does not correspond to the interface module Antrieb: Datenaufbau entspricht nicht Interface Mode'; 7515 'Drive: Power unit and motor incorrectly connected / Antrieb: Leistungsteil und Motor falsch verbunden'; 7516 'Drive: Re-commission the data set / Antrieb: Datensatz neu in Betrieb nehmen'; 7517 'Drive: Encoder data set changeover incorrectly parameterized / Antrieb: Geberdatensatzumschaltung falsch parametriert'; 7518 'Drive: Motor data set changeover incorrectly parameterized / Antrieb: Motordatensatzumschaltung falsch parametriert'; 7519 'Drive: Motor changeover incorrectly parameterized / Antrieb: Motorumschaltung falsch parametriert'; 7520 'Drive: Motor cannot be changed over / Antrieb: Motorumschaltung kann nicht ausgeführt werden'; 7530 'Drive: Drive Data Set DDS not present / Antrieb: Antriebsdatensatz DDS nicht vorhanden'; 7531 'Drive: Command Data Set CDS not present / Antrieb: Befehlsdatensatz CDS nicht vorhanden'; 7541 'Drive: Data set changeover not possible / Antrieb: Datensatzumschaltung nicht möglich'; 7545 'Drive: Pulse encoder interface parameterized incorrectly / Antrieb: WSG-Schnittstelle falsch parametriert'; 7550 'Drive: Not possible to reset encoder parameters / Antrieb: Geberparameter zurücksetzen nicht möglich'; 7551 'Drive encoder: No commutation angle information / Antrieb Geber: Keine Kommutierungswinkel-Information'; 7552 'Drive encoder: Encoder configuration not supported / Antrieb Geber: Geberkonfiguration nicht unterstützt'; 7553 'Drive encoder: Sensor Module configuration not supported / Antrieb Geber: Sensor Module Konfiguration nicht unterstützt'; 7555 'Drive encoder: Configuration position tracking / Antrieb Geber: Konfiguration Lageverfolgung'; 7556 'Measuring gear: Position tracking, maximum actual value exceeded Messgetriebe: Lageverfolgung maximaler Istwert überschritten'; 7557 'Encoder 1: Reference point coordinate not in the permissible range Geber 1: Referenzpunkt-Koordinate nicht im zulässigen Bereich'; 7558 'Encoder 2: Reference point coordinate not in the permissible range Geber 2: Referenzpunkt-Koordinate nicht im zulässigen Bereich'; 7559 'Encoder 3: Reference point coordinate not in the permissible range Geber 3: Referenzpunkt-Koordinate nicht im zulässigen Bereich'; 7560 'Drive encoder: Number of pulses is not to the power of two / Antrieb Geber: Strichzahl ist keine Zweierpotenz'; 7561 'Drive encoder: Number of multiturn pulses is not to the power of two Antrieb Geber: Strichzahl Multiturn keine Zweierpotenz'; 7562 'Drive, encoder: Position tracking, incremental encoder not possible Antrieb Geber: Lageverfolgung Inkrementalgeber nicht möglich'; 7565 'Drive: Encoder error in PROFIdrive encoder interface 1 / Antrieb: Geberfehler PROFIdrive-Geberschnittstelle 1'; 7566 'Drive: Encoder error in PROFIdrive encoder interface 2 / Antrieb: Geberfehler PROFIdrive-Geberschnittstelle 2'; 7567 'Drive: Encoder error in PROFIdrive encoder interface 3 / Antrieb: Geberfehler PROFIdrive-Geberschnittstelle 3'; 7569 'Encoder could not be identified / Geber konnte nicht identifiziert werden'; 7575 'Drive: Motor encoder not ready / Antrieb: Motorgeber nicht bereit'; 7576 'Drive: Encoderless operation due to a fault active / Antrieb: Geberloser Betrieb aufgrund Störung aktiv'; 7577 'Encoder 1: Measuring probe evaluation not possible / Geber 1: Messtasterauswertung nicht möglich'; 7578 'Encoder 2: Measuring probe evaluation not possible / Geber 2: Messtasterauswertung nicht möglich'; 7579 'Encoder 3: Measuring probe evaluation not possible / Geber 3: Messtasterauswertung nicht möglich'; 7580 'Drive: No Sensor Module with matching component number Antrieb: Kein Sensor Module mit passender Komponentennummer'; 7581 'Encoder 1: Position actual value preprocessing error / Geber 1: Lageistwertaufbereitung fehlerhaft'; 7582 'Encoder 2: Position actual value preprocessing error / Geber 2: Lageistwertaufbereitung fehlerhaft'; 7583 'Encoder 3: Position actual value preprocessing error / Geber 3: Lageistwertaufbereitung fehlerhaft'; 7584 'Encoder 1: Position setting value activated / Geber 1: Lagesetzwert aktiviert'; 7585 'Encoder 2: Position setting value activated / Geber 2: Lagesetzwert aktiviert'; 7586 'Encoder 3: Position setting value activated / Geber 3: Lagesetzwert aktiviert'; 7587 'Encoder 1: Position actual value preprocessing does not have a valid encoder Geber 1: Lageistwertaufbereitung hat keinen gültigen Geber'; 7588 'Encoder 2: Position actual value preprocessing does not have a valid encoder Geber 2: Lageistwertaufbereitung hat keinen gültigen Geber'; 7589 'Encoder 3: Position actual value preprocessing does not have a valid encoder Geber 3: Lageistwertaufbereitung hat keinen gültigen Geber'; 7590 'Encoder 1: Drive Data Set changeover in operation / Geber 1: Antriebsdatensatz-Umschaltung während Betrieb'; 7591 'Encoder 2: Drive Data Set changeover in operation / Geber 2: Antriebsdatensatz-Umschaltung während Betrieb'; 7592 'Encoder 3: Drive Data Set changeover in operation / Geber 3: Antriebsdatensatz-Umschaltung während Betrieb'; 7593 'Encoder 1: Value range for position actual value exceeded / Geber 1: Wertebereich für Lageistwert überschritten'; 7594 'Encoder 2: Value range for position actual value exceeded / Geber 2: Wertebereich für Lageistwert überschritten'; 7595 'Encoder 3: Value range for position actual value exceeded / Geber 3: Wertebereich für Lageistwert überschritten'; 7596 'Encoder 1: Reference function interrupted / Geber 1: Referenzfunktion abgebrochen'; 7597 'Encoder 2: Reference function interrupted / Geber 2: Referenzfunktion abgebrochen'; 7598 'Encoder 3: Reference function interrupted / Geber 3: Referenzfunktion abgebrochen'; 7599 'Encoder 1: Adjustment not possible / Geber 1: Justage nicht möglich'; 7600 'Encoder 2: Adjustment not possible / Geber 2: Justage nicht möglich'; 7601 'Encoder 3: Adjustment not possible / Geber 3: Justage nicht möglich'; 7800 'Drive: No power unit present / Antrieb: Kein Leistungsteil vorhanden'; 7801 'Drive: Motor overcurrent / Antrieb: Motor Überstrom'; 7802 'Drive: Infeed or power unit not ready / Antrieb: Einspeisung oder Leistungsteil nicht bereit'; 7805 'Drive: Power unit overload I2t / Antrieb: Leistungsteil Überlastung I2t'; 7806 'Drive: Regenerative power limit exceeded (F3E) / Antrieb: Generatorische Leistungsgrenze überschritten (F3E)'; 7807 'Drive: Short-circuit detected / Antrieb: Kurzschluss erkannt'; 7808 'HF damping module: damping not ready / HF Dämpfungsmodul: Dämpfung nicht bereit'; 7810 'Drive: Power unit EEPROM without rated data / Antrieb: Leistungsteil-EEPROM ohne Nenndaten'; 7815 'Drive: Power unit has been changed / Antrieb: Leistungsteil wurde geändert'; 7820 'Drive: Temperature sensor not connected / Antrieb: Temperatursensor nicht angeschlossen'; 7825 'Drive: Simulation mode activated / Antrieb: Simulationsbetrieb aktiviert'; 7826 'Drive: DC link voltage for simulation operation too high / Antrieb: Zwischenkreisspannung bei Simulationsbetrieb zu hoch'; 7840 'Drive: Infeed operation missing / Antrieb: Einspeisung Betrieb fehlt'; 7841 'Drive: Infeed operation withdrawn / Antrieb: Einspeisung Betrieb zurückgenommen'; 7850 'External alarm 1 / Externe Warnung 1'; 7851 'External alarm 2 / Externe Warnung 2'; 7852 'External alarm 3 / Externe Warnung 3'; 7860 'External fault 1 / Externe Störung 1'; 7861 'External fault 2 / Externe Störung 2'; 7862 'External fault 3 / Externe Störung 3'; 7890 'Internal voltage protection / internal armature short-circuit with STO active Interner Spannungsschutz/Interner Ankerkurzschluss mit STO aktiv'; 7900 'Drive: Motor blocked / Antrieb: Motor blockiert'; 7901 'Drive: Motor overspeed / Antrieb: Motor Überdrehzahl'; 7902 'Drive: Motor stalled / Antrieb: Motor gekippt'; 7903 'Drive: Motor speed deviation / Antrieb: Motor Drehzahlabweichung'; 7904 'External armature short-circuit: Contactor feedback signal 'Closed' missing Ankerkurzschluss extern: Schützrückmeldung 'Geschlossen' fehlt'; 7905 'External armature short-circuit: Contactor feedback signal 'Open' missing Ankerkurzschluss extern: Schützrückmeldung 'Offen' fehlt'; 7906 'Armature short-circuit / internal voltage protection: Parameterization error Ankerkurzschluss/Spannungsschutz intern: Parametrierung fehlerhaft'; 7907 'Internal armature short-circuit: Motor terminals are not at zero potential after pulse suppression Interner Ankerkurzschluss: Motorklemmen nach Impulslöschung nicht potenzialfrei'; 7908 'Internal armature short-circuit active / Interner Ankerkurzschluss aktiv'; 7909 'Internal voltage protection: De-activation only effective after POWER ON Interner Spannungsschutz: Deaktivierung erst nach POWER ON wirksam'; 7910 'Drive: Motor overtemperature / Antrieb: Motor Übertemperatur'; 7913 'Excitation current outside the tolerance range / Erregerstrom außerhalb Toleranz'; 7914 'Flux out of tolerance / Fluss außerhalb Toleranz'; 7918 'Three-phase setpoint generator operation selected/active / Drehstromsollwertgeberbetrieb angewählt/aktiv'; 7920 'Drive: Torque/speed too low / Antrieb: Drehmoment/Drehzahl zu niedrig'; 7921 'Drive: Torque/speed too high / Antrieb: Drehmoment/Drehzahl zu hoch'; 7922 'Drive: Torque/speed out of tolerance / Antrieb: Drehmoment/Drehzahl außerhalb Toleranz'; 7923 'Drive: Torque/speed too low / Antrieb: Drehmoment/Drehzahl zu niedrig'; 7924 'Drive: Torque/speed too high / Antrieb: Drehmoment/Drehzahl zu hoch'; 7925 'Drive: Torque/speed out of tolerance / Antrieb: Drehmoment/Drehzahl außerhalb Toleranz'; 7926 'Drive: Envelope curve, parameter invalid / Antrieb: Hüllkurve Parameter ungültig'; 7927 'DC braking active / Gleichstrombremsung aktiv'; 7928 'Internal voltage protection initiated / Interner Spannungsschutz ausgelöst'; 7929 'Drive: No motor detected / Antrieb: Kein Motor erkannt'; 7930 'Drive: Brake control error / Antrieb: Bremsenansteuerung fehlerhaft'; 7931 'Brake does not open / Bremse öffnet nicht'; 7932 'Brake does not close / Bremse schließt nicht'; 7934 'Drive: S120 Combi motor holding brake configuration / Antrieb: S120 Combi Motorhaltebremse Konfiguration'; 7935 'Drv: Motor holding brake detected / Antrieb: Motorhaltebremse erkannt'; 7936 'Drive: load failure / Antrieb: Lastausfall'; 7937 'Drive: Speed deviation between motor model and external speed Antrieb: Drehzahlabweichung Motormodell zu externer Drehzahl'; 7950 'Motor parameter incorrect / Motorparameter fehlerhaft'; 7955 'Drive: Motor has been changed / Antrieb: Motor wurde geändert'; 7956 'Drive: Motor code does not match the list (catalog) motor / Antrieb: Motorcode zum Listenmotor nicht passend'; 7960 'Drive: Incorrect friction characteristic / Antrieb: Reibkennlinie fehlerhaft'; 7961 'Drive: Friction characteristic record activated / Antrieb: Reibkennlinie Record aktiviert'; 7963 'Drive: Friction characteristic record interrupted / Antrieb: Reibkennlinie Record abgebrochen'; 7965 'Drive: Save required / Antrieb: Speichern erforderlich'; 7966 'Drive: Check the commutation angle / Antrieb: Kommutierungswinkel prüfen'; 7967 'Drive: Pole position identification internal fault / Antrieb: Pollageidentifikation interner Fehler'; 7968 'Drive: Lq-Ld measurement incorrect / Antrieb: Lq-Ld-Messung fehlerhaft'; 7969 'Drive: Incorrect pole position identification / Antrieb: Pollageidentifikation fehlerhaft'; 7970 'Drive: Automatic encoder adjustment incorrect / Antrieb: Automatische Geberjustage fehlerhaft'; 7971 'Drive: Angular commutation offset determination activated / Antrieb: Kommutierungswinkeloffset Ermittlung aktiviert'; 7980 'Drive: Rotating measurement activated / Antrieb: Drehende Messung aktiviert'; 7981 'Drive: Enable signals for the rotating measurement missing / Antrieb: Drehende Messung Freigaben fehlen'; 7982 'Drive: Rotating measurement encoder test / Antrieb: Drehende Messung Gebertest'; 7983 'Drive: Rotating measurement saturation characteristic / Antrieb: Drehende Messung Sättigungskennlinie'; 7984 'Drive: Speed controller optimization, moment of inertia / Antrieb: Drehzahlregleroptimierung Trägheitsmoment'; 7985 'Drive: Speed controller optimization (oscillation test) / Antrieb: Drehzahlregleroptimierung (Schwingungstest)'; 7986 'Drive: Rotating measurement ramp-function generator / Antrieb: Drehende Messung Hochlaufgeber'; 7987 'Drive: Rotating measurement, no encoder available / Antrieb: Drehende Messung Kein Geber verfügbar'; 7988 'Drive: Rotating measurement, no configuration selected / Antrieb: Drehende Messung Keine Konfiguration ausgewählt'; 7989 'Drive: Rotating measurement leakage inductance (q-axis) / Antrieb: Drehende Messung Streuinduktivität (q-Richtung)'; 7990 'Drive: Incorrect motor data identification / Antrieb: Motordatenidentifikation fehlerhaft'; 7991 'Drive: Motor data identification activated / Antrieb: Motordatenidentifikation aktiviert'; 7993 'Drive: Incorrect direction of rotation of the field or encoder actual value inversion Antrieb: Drehfeldrichtung oder Geberistwertinvertierung falsch'; 7994 'Drive: motor data identification not performed / Antrieb: Motordatenidentifikation nicht durchgeführt'; 7995 'Drive: Pole position identification not successful / Antrieb: Pollageidentifikation fehlgeschlagen'; 7996 'Drive: Pole position identification routine not carried out / Antrieb: Pollageidentifikation nicht erfolgt'; 7997 'Drive: Motor data identification active on another drive / Antrieb: Motordatenidentifikation auf anderem Antrieb aktiv'; 7998 'Drive: Motor data identification active on another drive / Antrieb: Motordatenidentifikation auf anderem Antrieb aktiv'; 7999 'Drive: Motor data identification cannot be activated / Antrieb: Motordatenidentifikation kann nicht aktiviert werden'; 8000 'TB: +/-15 V power supply faulted / TB: Versorgungsspannung +/-15 V fehlerhaft'; 8010 'CU: Analog-to-digital converter / CU: Analog-Digital-Wandler'; 8500 'COMM BOARD: Monitoring time configuration expired / COMM BOARD: Überwachungszeit Konfiguration abgelaufen'; 8501 'COMM BOARD: Setpoint timeout / COMM BOARD: Sollwert Timeout'; 8502 'COMM BOARD: Monitoring time sign-of-life expired / COMM BOARD: Überwachungszeit Lebenszeichen abgelaufen'; 8503 'COMM BOARD: Monitoring time non-cyclic channel expired COMM BOARD: Überwachungszeit azyklischer Kanal abgelaufen'; 8504 'COMM BOARD: Internal cyclic data transfer error COMM BOARD: Interner Fehler bei zyklischer Datenübertragung'; 8510 'COMM BOARD: Send configuration data invalid / COMM BOARD: Sende-Konfigurationsdaten ungültig'; 8511 'COMM BOARD: Receive configuration data invalid / COMM BOARD: Empfangs-Konfigurationsdaten ungültig'; 8520 'COMM BOARD: Non-cyclic channel error / COMM BOARD: Azyklischer Kanal fehlerhaft'; 8525 'COMM BOARD: Cyclic channel synchronization / COMM BOARD: Zyklischer Kanal Synchronisation'; 8526 'COMM BOARD: No cyclic connection / COMM BOARD: Keine zyklische Verbindung'; 8530 'COMM BOARD: Message channel error / COMM BOARD: Meldungskanal fehlerhaft'; 8550 'PZD Interface Hardware assignment error / PZD Interface Hardware-Zuordnung fehlerhaft'; 8560 'IE: Syntax error in configuration file / IE: Syntaxfehler in Konfigurationsdatei'; 8561 'IE: Consistency error affecting adjustable parameters / IE: Konsistenzfehler bei Einstellparametern'; 8562 'PN: Syntax error in configuration file / PN: Syntaxfehler in Konfigurationsdatei'; 8563 'PN: Consistency error affecting adjustable parameters / PN: Konsistenzfehler bei Einstellparametern'; 8564 'CBE20: Syntax error in configuration file / CBE20: Syntaxfehler in Konfigurationsdatei'; 8565 'CBE20: Consistency error affecting adjustable parameters / CBE20: Konsistenzfehler bei Einstellparametern'; 8700 'CAN: Communications error / CAN: Kommunikation fehlerhaft'; 8701 'CAN: NMT state change / CAN: NMT Zustandswechsel'; 8702 'CAN: RPDO Timeout'; 8703 'CAN: Maximum number of drive objects exceeded / CAN: Maximale Anzahl von Antriebsobjekten überschritten'; 8751 'CAN: Telegram loss / CAN: Telegrammverlust'; 8752 'CAN: Error counter for error passive exceeded / CAN: Fehlerzähler für Error Passive überschritten'; 8753 'CAN: Message buffer overflow / CAN: Nachrichtenpuffer übergelaufen'; 8754 'CAN: Incorrect communications mode / CAN: Kommunikationsmodus falsch'; 8755 'CAN: Obj cannot be mapped / CAN: Objekt nicht mappbar'; 8756 'CAN: Number of mapped bytes exceeded / CAN: Anzahl gemappte Bytes überschritten'; 8757 'CAN: Set COB-ID invalid / CAN: COB-ID ungültig setzen'; 8758 'CAN: Number of PDO channels too low / CAN: Anzahl PDO-Kanäle zu klein'; 8759 'CAN: PDO COB-ID already available / CAN: PDO COB-ID bereits vorhanden'; 13000 'License not adequate / Lizenzierung nicht ausreichend'; 13001 'Error in license checksum / Lizenzierung Prüfsumme fehlerhaft'; 13009 'Licensing OA application not licensed / Lizenzierung OA-Applikation nicht lizenziert'; 13010 'Licensing function module not licensed / Lizenzierung Funktionsmodul nicht lizenziert'; 13020 'Licensing not sufficient in the control / Lizenzierung nicht ausreichend in Steuerung'; 30001 'Power unit: Overcurrent / Leistungsteil: Überstrom'; 30002 'Power unit: DC link voltage, overvoltage / Leistungsteil: Zwischenkreisspannung Überspannung'; 30003 'Power unit: DC link voltage, undervoltage / Leistungsteil: Zwischenkreisspannung Unterspannung'; 30004 'Power unit: Overtemperature heat sink AC inverter / Leistungsteil: Übertemperatur Kühlkörper Wechselrichter'; 30005 'Power unit: Overload I2t / Leistungsteil: Überlastung I2t'; 30006 'Power unit: Thyristor Control Board / Leistungsteil: Thyristor Control Board'; 30008 'Power unit: Sign-of-life error cyclic data / Leistungsteil: Lebenszeichenfehler zyklische Daten'; 30010 'Power unit: Sign-of-life error cyclic data / Leistungsteil: Lebenszeichenfehler zyklische Daten'; 30011 'Power unit: Line phase failure in main circuit / Leistungsteil: Netzphasenausfall im Hauptstromkreis'; 30012 'Power unit: Temperature sensor heat sink wire breakage / Leistungsteil: Temperaturfühler Kühlkörper Drahtbruch'; 30013 'Power unit: Temperature sensor heat sink short-circuit / Leistungsteil: Temperaturfühler Kühlkörper Kurzschluss'; 30015 'Power unit: Phase failure motor cable / Leistungsteil: Phasenausfall Motorleitung'; 30016 'Power unit: Load supply switched out / Leistungsteil: Lastversorgung ausgeschaltet'; 30017 'Power unit: Hardware current limit has responded too often / Leistungsteil: Hardware Strombegrenzung zu oft angesprochen'; 30020 'Power unit: Configuration not supported / Leistungsteil: Konfiguration nicht unterstützt'; 30021 'Power unit: Ground fault / Leistungsteil: Erdschluss'; 30022 'Power unit: Monitoring U_ce / Leistungsteil: Überwachung U_ce'; 30023 'Power unit: Overtemperature thermal model alarm / Leistungsteil: Übertemperatur Thermisches Modell Warnung'; 30024 'Power unit: Overtemperature thermal model / Leistungsteil: Übertemperatur Thermisches Modell'; 30025 'Power unit: Chip overtemperature / Leistungsteil: Übertemperatur Chip'; 30027 'Power unit: Precharging DC link time monitoring / Leistungsteil: Vorladung Zwischenkreis Zeitüberwachung'; 30031 'Power unit: Hardware current limiting, phase U / Leistungsteil: Hardware Strombegrenzung in Phase U'; 30032 'Power unit: Hardware current limiting, phase V / Leistungsteil: Hardware Strombegrenzung in Phase V'; 30033 'Power unit: Hardware current limiting, phase W / Leistungsteil: Hardware Strombegrenzung in Phase W'; 30034 'Power unit: Internal overtemperature / Leistungsteil: Übertemperatur Innenraum'; 30035 'Power unit: Air intake overtemperature / Leistungsteil: Übertemperatur Zuluft'; 30036 'Power unit: Internal overtemperature / Leistungsteil: Übertemperatur Innenraum'; 30037 'Power unit: Rectifier overtemperature / Leistungsteil: Übertemperatur Gleichrichter'; 30040 'Undervoltage 24 V / Unterspannung 24 V'; 30041 'Undervoltage 24 V alarm / Unterspannung 24 V Warnung'; 30042 'Power unit: Fan operating time reached or exceeded / Leistungsteil: Betriebsdauer Lüfter erreicht oder überschritten'; 30043 '24 V overvoltage / Überspannung 24 V'; 30044 'Overvoltage 24 V alarm / Überspannung 24 V Warnung'; 30045 'Power unit: Supply undervoltage / Leistungsteil: Unterspannung Versorgung'; 30046 'Power unit: Undervoltage, alarm / Leistungsteil: Unterspannung Warnung'; 30048 'Power unit: External fan faulty / Leistungsteil: Externer Lüfter defekt'; 30049 'Power unit: Internal fan faulty / Leistungsteil: Innenraumlüfter defekt'; 30050 'Power unit: 24 V supply overvoltage / Leistungsteil: Überspannung 24-V-Versorgung'; 30052 'EEPROM data error / EEPROM Daten fehlerhaft'; 30053 'FPGA data faulty / FPGA Daten fehlerhaft'; 30054 'Power unit: Undervoltage when opening the brake / Leistungsteil: Unterspannung bei Bremse öffnen'; 30055 'Power unit: Braking chopper overcurrent / Leistungsteil: Bremschopper Überstrom'; 30059 'Power unit: Internal fan faulty / Leistungsteil: Innenraumlüfter defekt'; 30060 'Pre-charge contactor state monitoring / Vorladeschütz Zustandsüberwachung'; 30061 'Bypass contactor monitoring / Überbrückungsschütz Zustandsüberwachung'; 30070 'Cycle requested by the power unit module not supported Angeforderter Zyklus von Leistungsteilbaugruppe nicht unterstützt'; 30071 'No new actual values received from the Power Module / Keine neuen Istwerte von Power Module empfangen'; 30072 'Setpoints can no longer be transferred to the Power Module / Keine Sollwerte mehr an Power Module übertragbar'; 30073 'Actual value/setpoint preprocessing no longer synchronous / Istwert-/Sollwertaufbereitung nicht mehr synchron'; 30074 'Communication error between the Control Unit and Power Module Kommunikationsfehler zwischen Control Unit und Power Module'; 30080 'Power unit: Current increasing too quickly / Leistungsteil: Stromanstieg zu schnell'; 30081 'Power unit: Switching operations too frequent / Leistungsteil: Schalthandlungen zu häufig'; 30105 'PU: Actual value sensing fault / LT: Istwerterfassung fehlerhaft'; 30314 'Power unit: 24 V power supply overloaded by PM / Leistungsteil: 24-V-Versorgung über PM überlastet'; 30315 'Power unit: 24 V power supply overloaded by PM / Leistungsteil: 24-V-Versorgung über PM überlastet'; 30502 'Power unit: DC link overvoltage / Leistungsteil: Zwischenkreis Überspannung'; 30600 'SI P2: STOP A initiated / SI P2: STOP A ausgelöst'; 30611 'SI P2: Defect in a monitoring channel / SI P2: Defekt in einem Überwachungskanal'; 30620 'SI P2: Safe Torque Off active / SI P2: Sicher abgeschaltetes Moment aktiv'; 30621 'SI MM: Safe Stop 1 active / SI MM: Safe Stop 1 aktiv'; 30625 'SI P2: Sign-of-life error in safety data / SI P2: Lebenszeichen in Safety-Daten fehlerhaft'; 30630 'SI MM: Brake control error / SI MM: Bremsenansteuerung fehlerhaft'; 30640 'SI MM: Fault in the shutdown path of the second channel / SI MM: Fehler im Abschaltpfad des zweiten Kanals'; 30649 'SI MM / P2: Internal software error / SI MM / P2: Softwarefehler intern'; 30650 'SI MM / P2: Acceptance test required / SI MM / P2: Abnahmetest erforderlich'; 30651 'SI MM / P2: Synchronization with Control Unit unsuccessful / SI MM / P2: Synchronisation mit Control Unit fehlgeschlagen'; 30652 'SI MM: Illegal monitoring clock cycle / SI MM: Überwachungstakt unzulässig'; 30655 'SI MM / P2: Align monitoring functions / SI MM / P2: Abgleich der Überwachungsfunktionen'; 30656 'SI MM / P2: Motor Module parameter error / SI MM / P2: Parameter Motor Module fehlerhaft'; 30659 'SI MM / P2: Write request for parameter rejected / SI MM / P2: Schreibauftrag für Parameter abgewiesen'; 30662 'Error in internal communications / Fehler in interner Kommunikation'; 30664 'Error while booting / Fehler in der Hochlaufphase'; 30665 'SI MM / P2: System is defective / SI MM / P2: System ist defekt'; 30666 'SI Motion MM / P2: Steady-state (static) 1 signal at the F-DI for safety-relevant acknowledgement SI Motion MM / P2: Statisches 1-Signal am F-DI für sichere Quittierung'; 30672 'SI CU: Control Unit software incompatible / SI CU: Control Unit Software inkompatibel'; 30680 'SI Motion MM / P2: Checksum error safety monitoring functions / SI Motion MM / P2: Prüfsummenfehler sichere Überwachungen'; 30681 'SI Motion MM / P2: Incorrect parameter value / SI Motion MM / P2: Parameterwert falsch'; 30682 'SI Motion MM / P2: Monitoring function not supported / SI Motion MM / P2: Überwachungsfunktion nicht unterstützt'; 30683 'SI Motion MM / P2: SOS/SLS enable missing / SI Motion MM / P2: SOS/SLS-Freigabe fehlt'; 30685 'SI Motion MM: Safely-Limited Speed limit value too high SI Motion MM: Sicher begrenzte Geschwindigkeit Grenzwert zu groß'; 30688 'SI Motion MM: Actual value synchronization not permissible / SI Motion MM: Istwertsynchronisation nicht zulässig'; 30692 'SI Motion MM / P2: Incorrect parameter value encoderless / SI Motion MM / P2: Parameterwert falsch geberlos'; 30693 'SI MM / P2: Safety parameter settings changed, warm restart/POWER ON required SI MM / P2: Safety-Parametrierung geändert Warmstart/POWER ON erforderlich'; 30700 'SI Motion MM / P2: STOP A initiated / SI Motion MM / P2: STOP A ausgelöst'; 30701 'SI Motion MM / P2: STOP B initiated / SI Motion MM / P2: STOP B ausgelöst'; 30706 'SI Motion MM / P2: SAM/SBR limit exceeded / SI Motion MM / P2: SAM/SBR Grenze überschritten'; 30707 'SI Motion MM: Tolerance for safe operating stop exceeded / SI Motion MM: Toleranz für Sicheren Betriebshalt überschritten'; 30708 'SI Motion MM: STOP C initiated / SI Motion MM: STOP C ausgelöst'; 30709 'SI Motion MM: STOP D initiated / SI Motion MM: STOP D ausgelöst'; 30710 'SI Motion MM: STOP E initiated / SI Motion MM: STOP E ausgelöst'; 30711 'SI Motion MM / P2: Defect in a monitoring channel / SI Motion MM / P2: Defekt in einem Überwachungskanal'; 30712 'SI Motion MM / P2: Defect in F-IO processing / SI Motion MM / P2: Defekt bei F-IO-Verarbeitung'; 30714 'SI Motion MM / P2: Safely-Limited Speed exceeded SI Motion MM / P2: Sicher begrenzte Geschwindigkeit überschritten'; 30716 'SI Motion MM / P2: Tolerance for safe motion direction exceeded SI Motion MM / P2: Toleranz für sichere Bewegungsrichtung überschritten'; 30770 'SI Motion MM / P2: Discrepancy error affecting the fail-safe inputs/outputs SI Motion MM / P2: Diskrepanzfehler der fehlersicheren Eingänge/Ausgänge'; 30772 'SI Motion MM: Test stop failsafe inputs/outputs active SI Motion MM: Teststop fehlersichere Eingänge/Ausgänge aktiv'; 30773 'SI Motion MM: Test stop fault Motor Module / SI Motion MM: Teststop fehlerhaft Motor Module'; 30798 'SI Motion MM / P2: Test stop running / SI Motion MM / P2: Teststop läuft'; 30799 'SI Motion MM / P2: Acceptance test mode active / SI Motion MM / P2: Abnahmetestmodus aktiv'; 30800 'Power unit: Group signal / Leistungsteil: Sammelmeldung'; 30802 'Power unit: Time slice overflow / Leistungsteil: Zeitscheibenüberlauf'; 30804 'Power unit: CRC / Leistungsteil: CRC'; 30805 'Power unit: EPROM checksum error / Leistungsteil: Prüfsumme EPROM nicht korrekt'; 30809 'Power unit: Switching information not valid / Leistungsteil: Schaltinformation ungültig'; 30810 'Power unit: Watchdog timer / Leistungsteil: Watchdog Timer'; 30850 'Power unit: Internal software error / Leistungsteil: Softwarefehler intern'; 30853 'Power unit: Sign-of-life error cyclic data / Leistungsteil: Lebenszeichenfehler zyklische Daten'; 30898 'Power unit: POWER ON signal / Leistungsteil: POWER ON Meldung'; 30899 'Power unit: Unknown fault / Leistungsteil: Unbekannte Störung'; 30903 'Power unit: I2C bus error occurred / Leistungsteil: I2C-Bus Fehler aufgetreten'; 30907 'Power unit: FPGA configuration unsuccessful / Leistungsteil: FPGA-Konfiguration fehlgeschlagen'; 30920 'Temperature sensor fault / Fehler Temperatursensor'; 30999 'Power unit: Unknown alarm / Leistungsteil: Unbekannte Warnung'; 31100 'Encoder 1: Zero mark distance error / Geber 1: Nullmarkenabstand fehlerhaft'; 31101 'Encoder 1: Zero mark failed / Geber 1: Nullmarke ausgefallen'; 31103 'Encoder 1: Amplitude error, track R / Geber 1: Amplitudenfehler Spur R'; 31110 'Encoder 1: Serial communications error / Geber 1: Serielle Kommunikation gestört'; 31111 'Encoder 1: Absolute encoder EnDat, internal fault/error / Geber 1: Absolutwertgeber EnDat interner Fehler'; 31112 'Encoder 1: Error bit set in the serial protocol / Geber 1: Fehlerbit im seriellen Protokoll gesetzt'; 31115 'Encoder 1: Amplitude error track A or B (A^2 + B^2) / Geber 1: Amplitudenfehler Spur A oder B (A^2 + B^2)'; 31116 'Encoder 1: Amplitude error monitoring track A + B / Geber 1: Amplitudenfehler Überwachung Spur A + B'; 31117 'Encoder 1: Inversion error signals A/B/R / Geber 1: Invertierung Signal A/B/R fehlerhaft'; 31118 'Encoder 1: Speed difference outside the tolerance range / Geber 1: Drehzahldifferenz außerhalb Toleranz'; 31120 'Encoder 1: Power supply voltage fault / Geber 1: Versorgungsspannung fehlerhaft'; 31121 'Encoder 1: Coarse position error / Geber 1: Groblage fehlerhaft'; 31122 'Encoder 1: Internal power supply voltage faulty / Geber 1: Interne Versorgungsspannung fehlerhaft'; 31123 'Encoder 1: Signal level A/B unipolar outside tolerance / Geber 1: Signalpegel A/B unipolar außerhalb Toleranz'; 31125 'Encoder 1: Amplitude error track A or B overcontrolled / Geber 1: Amplitudenfehler Spur A oder B übersteuert'; 31126 'Encoder 1: Amplitude AB too high / Geber 1: Amplitude AB zu hoch'; 31129 'Encoder 1: Position difference, hall sensor/track C/D and A/B too large Geber 1: Lagedifferenz Hallsensor/Spur C/D und Spur A/B zu groß'; 31130 'Encoder 1: Zero mark and position error from the coarse synchronization Geber 1: Nullmarke und Lage aus Grobsynchronisation falsch'; 31131 'Encoder 1: Deviation, position incremental/absolute too large / Geber 1: Abweichung Lage inkrementell/absolut zu groß'; 31135 'Encoder 1: Fault when determining the position / Geber 1: Fehler bei Lagebestimmung'; 31136 'Encoder 1: Error when determining multiturn information / Geber 1: Fehler bei Bestimmung der Multiturn-Information'; 31137 'Encoder 1: Internal fault when determining the position / Geber 1: Interner Fehler bei Lagebestimmung'; 31138 'Encoder 1: Internal error when determining multiturn information Geber 1: Interner Fehler bei Bestimmung der Multiturninformation'; 31150 'Encoder 1: Initialization error / Geber 1: Initialisierung fehlerhaft'; 31151 'Encoder 1: Encoder speed for initialization AB too high / Geber 1: Geberdrehzahl für Initialisierung zu hoch'; 31160 'Encoder 1: Analog sensor channel A failed / Geber 1: Analogsensor Kanal A ausgefallen'; 31161 'Encoder 1: Analog sensor channel B failed / Geber 1: Analogsensor Kanal B ausgefallen'; 31163 'Encoder 1: Analog sensor position value exceeds limit value / Geber 1: Analogsensor Lagewert überschreitet Grenzwert'; 31400 'Encoder 1: Alarm threshold zero mark distance error / Geber 1: Warnschwelle Nullmarkenabstand fehlerhaft'; 31401 'Encoder 1: Alarm threshold zero mark failed / Geber 1: Warnschwelle Nullmarke ausgefallen'; 31405 'Encoder 1: Temperature in the encoder evaluation inadmissible / Geber 1: Temperatur in Geberauswertung unzulässig'; 31407 'Encoder 1: Function limit reached / Geber 1: Funktionsgrenze erreicht'; 31410 'Encoder 1: Serial communications / Geber 1: Serielle Kommunikation'; 31411 'Encoder 1: EnDat encoder signals alarms / Geber 1: EnDat-Geber meldet Warnungen'; 31412 'Encoder 1: Error bit set in the serial protocol / Geber 1: Fehlerbit im seriellen Protokoll gesetzt'; 31414 'Encoder 1: Amplitude error track C or D (C^2 + D^2) / Geber 1: Amplitudenfehler Spur C oder D (C^2 + D^2)'; 31415 'Encoder 1: Amplitude alarm track A or B (A^2 + B^2) / Geber 1: Amplitudenwarnung Spur A oder B (A^2 + B^2)'; 31418 'Encoder 1: Speed difference per sampling rate exceeded / Geber 1: Drehzahldifferenz je Abtastrate überschritten'; 31419 'Encoder 1: Track A or B outside tolerance / Geber 1: Spur A oder B außerhalb Toleranz'; 31421 'Encoder 1: Coarse position error / Geber 1: Groblage fehlerhaft'; 31422 'Encoder 1: Pulses per revolution square-wave encoder outside tolerance bandwidth / Geber 1: Impulszahl Rechteckgeber außerhalb Toleranzband'; 31429 'Encoder 1: Position difference, hall sensor/track C/D and A/B too large Geber 1: Lagedifferenz Hallsensor/Spur C/D und Spur A/B zu groß'; 31431 'Encoder 1: Deviation, position incremental/absolute too large / Geber 1: Abweichung Lage inkrementell/absolut zu groß'; 31432 'Encoder 1: Rotor position adaptation corrects deviation / Geber 1: Rotorlageadaption korrigiert Abweichung'; 31442 'Encoder 1: Battery voltage pre-alarm / Geber 1: Batteriespannung Vorwarnung'; 31443 'Encoder 1: Unipolar CD signal level outside specification / Geber 1: Unipolar CD Signalpegel außerhalb Spezifikation'; 31460 'Encoder 1: Analog sensor channel A failed / Geber 1: Analogsensor Kanal A ausgefallen'; 31461 'Encoder 1: Analog sensor channel B failed / Geber 1: Analogsensor Kanal B ausgefallen'; 31462 'Encoder 1: Analog sensor, no channel active / Geber 1: Analogsensor Kein Kanal aktiv'; 31463 'Encoder 1: Analog sensor position value exceeds limit value / Geber 1: Analogsensor Lagewert überschreitet Grenzwert'; 31470 'Encoder 1: Soiling detected / Geber 1: Verschmutzung erkannt'; 31500 'Encoder 1: Position tracking traversing range exceeded / Geber 1: Lageverfolgung Verfahrbereich überschritten'; 31501 'Encoder 1: Position tracking encoder position outside tolerance window Geber 1: Lageverfolgung Geberposition außerhalb Toleranzfenster'; 31502 'Encoder 1: Encoder with measuring gear, without valid signals / Geber 1: Geber mit Messgetriebe ohne gültige Signale'; 31503 'Encoder 1: Position tracking cannot be reset / Geber 1: Lageverfolgung lässt sich nicht zurücksetzen'; 31700 'Encoder 1: Effectivity test does not supply the expected value / Geber 1: Wirksamkeitstest liefert nicht Erwartungswert'; 31800 'Encoder 1: Group signal / Geber 1: Sammelmeldung'; 31802 'Encoder 1: Time slice overflow / Geber 1: Zeitscheibenüberlauf'; 31804 'Encoder 1: Checksum error / Geber 1: Checksummenfehler'; 31805 'Encoder 1: EPROM checksum error / Geber 1: Prüfsumme EPROM nicht korrekt'; 31806 'Encoder 1: Initialization error / Geber 1: Initialisierung fehlgeschlagen'; 31811 'Encoder 1: Encoder serial number changed / Geber 1: Geberseriennummer geändert'; 31812 'Encoder 1: Requested cycle or RX-/TX timing not supported Geber 1: Angeforderter Zyklus bzw. RX-/TX-Timing nicht unterstützt'; 31813 'Encoder 1: Hardware logic unit failed / Geber 1: Hardware Logikeinheit ausgefallen'; 31850 'Encoder 1: Encoder evaluation, internal software error / Geber 1: Geberauswertung Softwarefehler intern'; 31898 'Encoder 1: POWER ON signal / Geber 1: POWER ON Meldung'; 31899 'Encoder 1: Unknown fault / Geber 1: Unbekannte Störung'; 31902 'Encoder 1: SPI-BUS error occurred / Geber 1: SPI-BUS Fehler aufgetreten'; 31903 'Encoder 1: I2C-BUS error occurred / Geber 1: I2C-BUS Fehler aufgetreten'; 31905 'Encoder 1: Parameterization error / Geber 1: Fehlparametrierung'; 31915 'Encoder 1: Configuration error / Geber 1: Konfigurationsfehler'; 31916 'Encoder 1: Parameterization fault / Geber 1: Fehler bei Parametrierung'; 31920 'Encoder 1: Temperature sensor fault / Geber 1: Fehler Temperatursensor'; 31930 'Encoder 1: Data logger has saved data / Geber 1: Datalogger hat Daten gespeichert'; 31940 'Sensor 1: Spindle clamping state error / Geber 1: Spindel Spannzustand fehlerhaft'; 31999 'Encoder 1: Unknown alarm / Geber 1: Unbekannte Warnung'; 32100 'Encoder 2: Zero mark distance error / Geber 2: Nullmarkenabstand fehlerhaft'; 32101 'Encoder 2: Zero mark failed / Geber 2: Nullmarke ausgefallen'; 32103 'Encoder 2: Amplitude error, track R / Geber 2: Amplitudenfehler Spur R'; 32110 'Encoder 2: Serial communications error / Geber 2: Serielle Kommunikation gestört'; 32111 'Encoder 2: Absolute encoder EnDat, internal fault/error / Geber 2: Absolutwertgeber EnDat interner Fehler'; 32112 'Encoder 2: Error bit set in the serial protocol / Geber 2: Fehlerbit im seriellen Protokoll gesetzt'; 32115 'Encoder 2: Amplitude error track A or B (A^2 + B^2) / Geber 2: Amplitudenfehler Spur A oder B (A^2 + B^2)'; 32116 'Encoder 2: Amplitude error monitoring track A + B / Geber 2: Amplitudenfehler Überwachung Spur A + B'; 32117 'Encoder 2: Inversion error signals A/B/R / Geber 2: Invertierung Signal A/B/R fehlerhaft'; 32118 'Encoder 2: Speed difference outside the tolerance range / Geber 2: Drehzahldifferenz außerhalb Toleranz'; 32120 'Encoder 2: Power supply voltage fault / Geber 2: Versorgungsspannung fehlerhaft'; 32121 'Encoder 2: Coarse position error / Geber 2: Groblage fehlerhaft'; 32122 'Encoder 2: Internal power supply voltage faulty / Geber 2: Interne Versorgungsspannung fehlerhaft'; 32123 'Encoder 2: Signal level A/B unipolar outside tolerance / Geber 2: Signalpegel A/B unipolar außerhalb Toleranz'; 32125 'Encoder 2: Amplitude error track A or B overcontrolled / Geber 2: Amplitudenfehler Spur A oder B übersteuert'; 32126 'Encoder 2: Amplitude AB too high / Geber 2: Amplitude AB zu hoch'; 32129 'Encoder 2: Position difference, hall sensor/track C/D and A/B too large Geber 2: Lagedifferenz Hallsensor/Spur C/D und Spur A/B zu groß'; 32130 'Encoder 2: Zero mark and position error from the coarse synchronization Geber 2: Nullmarke und Lage aus Grobsynchronisation falsch'; 32131 'Encoder 2: Deviation, position incremental/absolute too large / Geber 2: Abweichung Lage inkrementell/absolut zu groß'; 32135 'Encoder 2: Fault when determining the position / Geber 2: Fehler bei Lagebestimmung'; 32136 'Encoder 2: Error when determining multiturn information / Geber 2: Fehler bei Bestimmung der Multiturn-Information'; 32137 'Encoder 2: Internal fault when determining the position / Geber 2: Interner Fehler bei Lagebestimmung'; 32138 'Encoder 2: Internal error when determining multiturn information Geber 2: Interner Fehler bei Bestimmung der Multiturninformation'; 32150 'Encoder 2: Initialization error / Geber 2: Initialisierung fehlerhaft'; 32151 'Encoder 2: Encoder speed for initialization AB too high / Geber 2: Geberdrehzahl für Initialisierung zu hoch'; 32160 'Encoder 2: Analog sensor channel A failed / Geber 2: Analogsensor Kanal A ausgefallen'; 32161 'Encoder 2: Analog sensor channel B failed / Geber 2: Analogsensor Kanal B ausgefallen'; 32163 'Encoder 2: Analog sensor position value exceeds limit value / Geber 2: Analogsensor Lagewert überschreitet Grenzwert'; 32400 'Encoder 2: Alarm threshold zero mark distance error / Geber 2: Warnschwelle Nullmarkenabstand fehlerhaft'; 32401 'Encoder 2: Alarm threshold zero mark failed / Geber 2: Warnschwelle Nullmarke ausgefallen'; 32405 'Encoder 2: Temperature in the encoder evaluation inadmissible / Geber 2: Temperatur in Geberauswertung unzulässig'; 32407 'Encoder 2: Function limit reached / Geber 2: Funktionsgrenze erreicht'; 32410 'Encoder 2: Serial communications / Geber 2: Serielle Kommunikation'; 32411 'Encoder 2: EnDat encoder signals alarms / Geber 2: EnDat-Geber meldet Warnungen'; 32412 'Encoder 2: Error bit set in the serial protocol / Geber 2: Fehlerbit im seriellen Protokoll gesetzt'; 32414 'Encoder 2: Amplitude error track C or D (C^2 + D^2) / Geber 2: Amplitudenfehler Spur C oder D (C^2 + D^2)'; 32415 'Encoder 2: Amplitude alarm track A or B (A^2 + B^2) / Geber 2: Amplitudenwarnung Spur A oder B (A^2 + B^2)'; 32418 'Encoder 2: Speed difference per sampling rate exceeded / Geber 2: Drehzahldifferenz je Abtastrate überschritten'; 32419 'Encoder 2: Track A or B outside tolerance / Geber 2: Spur A oder B außerhalb Toleranz'; 32421 'Encoder 2: Coarse position error / Geber 2: Groblage fehlerhaft'; 32422 'Encoder 2: Pulses per revolution square-wave encoder outside tolerance bandwidth Geber 2: Impulszahl Rechteckgeber außerhalb Toleranzband'; 32429 'Encoder 2: Position difference, hall sensor/track C/D and A/B too large Geber 2: Lagedifferenz Hallsensor/Spur C/D und Spur A/B zu groß'; 32431 'Encoder 2: Deviation, position incremental/absolute too large / Geber 2: Abweichung Lage inkrementell/absolut zu groß'; 32432 'Encoder 2: Rotor position adaptation corrects deviation / Geber 2: Rotorlageadaption korrigiert Abweichung'; 32442 'Encoder 2: Battery voltage pre-alarm / Geber 2: Batteriespannung Vorwarnung'; 32443 'Encoder 2: Unipolar CD signal level outside specification / Geber 2: Unipolar CD Signalpegel außerhalb Spezifikation'; 32460 'Encoder 2: Analog sensor channel A failed / Geber 2: Analogsensor Kanal A ausgefallen'; 32461 'Encoder 2: Analog sensor channel B failed / Geber 2: Analogsensor Kanal B ausgefallen'; 32462 'Encoder 2: Analog sensor, no channel active / Geber 2: Analogsensor Kein Kanal aktiv'; 32463 'Encoder 2: Analog sensor position value exceeds limit value / Geber 2: Analogsensor Lagewert überschreitet Grenzwert'; 32470 'Encoder 2: Soiling detected / Geber 2: Verschmutzung erkannt'; 32500 'Encoder 2: Position tracking traversing range exceeded / Geber 2: Lageverfolgung Verfahrbereich überschritten'; 32501 'Encoder 2: Position tracking encoder position outside tolerance window Geber 2: Lageverfolgung Geberposition außerhalb Toleranzfenster'; 32502 'Encoder 2: Encoder with measuring gear, without valid signals / Geber 2: Geber mit Messgetriebe ohne gültige Signale'; 32503 'Encoder 2: Position tracking cannot be reset / Geber 2: Lageverfolgung lässt sich nicht zurücksetzen'; 32700 'Encoder 2: Effectivity test does not supply the expected value / Geber 2: Wirksamkeitstest liefert nicht Erwartungswert'; 32800 'Encoder 2: Group signal / Geber 2: Sammelmeldung'; 32802 'Encoder 2: Time slice overflow / Geber 2: Zeitscheibenüberlauf'; 32804 'Encoder 2: Checksum error / Geber 2: Checksummenfehler'; 32805 'Encoder 2: EPROM checksum error / Geber 2: Prüfsumme EPROM nicht korrekt'; 32806 'Encoder 2: Initialization error / Geber 2: Initialisierung fehlgeschlagen'; 32811 'Encoder 2: Encoder serial number changed / Geber 2: Geberseriennummer geändert'; 32812 'Encoder 2: Requested cycle or RX-/TX timing not supported Geber 2: Angeforderter Zyklus bzw. RX-/TX-Timing nicht unterstützt'; 32813 'Encoder 2: Hardware logic unit failed / Geber 2: Hardware Logikeinheit ausgefallen'; 32850 'Encoder 2: Encoder evaluation, internal software error / Geber 2: Geberauswertung Softwarefehler intern'; 32898 'Encoder 2: POWER ON signal / Geber 2: POWER ON Meldung'; 32899 'Encoder 2: Unknown fault / Geber 2: Unbekannte Störung'; 32902 'Encoder 2: SPI-BUS error occurred / Geber 2: SPI-BUS Fehler aufgetreten'; 32903 'Encoder 2: I2C-BUS error occurred / Geber 2: I2C-BUS Fehler aufgetreten'; 32905 'Encoder 2: Parameterization error / Geber 2: Fehlparametrierung'; 32915 'Encoder 2: Configuration error / Geber 2: Konfigurationsfehler'; 32916 'Encoder 2: Parameterization fault / Geber 2: Fehler bei Parametrierung'; 32920 'Encoder 2: Temperature sensor fault / Geber 2: Fehler Temperatursensor'; 32930 'Encoder 2: Data logger has saved data / Geber 2: Datalogger hat Daten gespeichert'; 32940 'Sensor 2: Spindle clamping state error / Geber 2: Spindel Spannzustand fehlerhaft'; 32999 'Encoder 2: Unknown alarm / Geber 2: Unbekannte Warnung'; 33100 'Encoder 3: Zero mark distance error / Geber 3: Nullmarkenabstand fehlerhaft'; 33101 'Encoder 3: Zero mark failed / Geber 3: Nullmarke ausgefallen'; 33103 'Encoder 3: Amplitude error, track R / Geber 3: Amplitudenfehler Spur R'; 33110 'Encoder 3: Serial communications error / Geber 3: Serielle Kommunikation gestört'; 33111 'Encoder 3: Absolute encoder EnDat, internal fault/error / Geber 3: Absolutwertgeber EnDat interner Fehler'; 33112 'Encoder 3: Error bit set in the serial protocol / Geber 3: Fehlerbit im seriellen Protokoll gesetzt'; 33115 'Encoder 3: Amplitude error track A or B (A^2 + B^2) / Geber 3: Amplitudenfehler Spur A oder B (A^2 + B^2)'; 33116 'Encoder 3: Amplitude error monitoring track A + B / Geber 3: Amplitudenfehler Überwachung Spur A + B'; 33117 'Encoder 3: Inversion error signals A/B/R / Geber 3: Invertierung Signal A/B/R fehlerhaft'; 33118 'Encoder 3: Speed difference outside the tolerance range / Geber 3: Drehzahldifferenz außerhalb Toleranz'; 33120 'Encoder 3: Power supply voltage fault / Geber 3: Versorgungsspannung fehlerhaft'; 33121 'Encoder 3: Coarse position error / Geber 3: Groblage fehlerhaft'; 33122 'Encoder 3: Internal power supply voltage faulty / Geber 3: Interne Versorgungsspannung fehlerhaft'; 33123 'Encoder 3: Signal level A/B unipolar outside tolerance / Geber 3: Signalpegel A/B unipolar außerhalb Toleranz'; 33125 'Encoder 3: Amplitude error track A or B overcontrolled / Geber 3: Amplitudenfehler Spur A oder B übersteuert'; 33126 'Encoder 3: Amplitude AB too high / Geber 3: Amplitude AB zu hoch'; 33129 'Encoder 3: Position difference, hall sensor/track C/D and A/B too large Geber 3: Lagedifferenz Hallsensor/Spur C/D und Spur A/B zu groß'; 33130 'Encoder 3: Zero mark and position error from the coarse synchronization Geber 3: Nullmarke und Lage aus Grobsynchronisation falsch'; 33131 'Encoder 3: Deviation, position incremental/absolute too large / Geber 3: Abweichung Lage inkrementell/absolut zu groß'; 33135 'Encoder 3: Fault when determining the position / Geber 3: Fehler bei Lagebestimmung'; 33136 'Encoder 3: Error when determining multiturn information / Geber 3: Fehler bei Bestimmung der Multiturn-Information'; 33137 'Encoder 3: Internal fault when determining the position / Geber 3: Interner Fehler bei Lagebestimmung'; 33138 'Encoder 3: Internal error when determining multiturn information Geber 3: Interner Fehler bei Bestimmung der Multiturninformation'; 33150 'Encoder 3: Initialization error / Geber 3: Initialisierung fehlerhaft'; 33151 'Encoder 3: Encoder speed for initialization AB too high / Geber 3: Geberdrehzahl für Initialisierung zu hoch'; 33160 'Encoder 3: Analog sensor channel A failed / Geber 3: Analogsensor Kanal A ausgefallen'; 33161 'Encoder 3: Analog sensor channel B failed / Geber 3: Analogsensor Kanal B ausgefallen'; 33163 'Encoder 3: Analog sensor position value exceeds limit value / Geber 3: Analogsensor Lagewert überschreitet Grenzwert'; 33400 'Encoder 3: Alarm threshold zero mark distance error / Geber 3: Warnschwelle Nullmarkenabstand fehlerhaft'; 33401 'Encoder 3: Alarm threshold zero mark failed / Geber 3: Warnschwelle Nullmarke ausgefallen'; 33405 'Encoder 3: Temperature in the encoder evaluation inadmissible / Geber 3: Temperatur in Geberauswertung unzulässig'; 33407 'Encoder 3: Function limit reached / Geber 3: Funktionsgrenze erreicht'; 33410 'Encoder 3: Serial communications / Geber 3: Serielle Kommunikation'; 33411 'Encoder 3: EnDat encoder signals alarms / Geber 3: EnDat-Geber meldet Warnungen'; 33412 'Encoder 3: Error bit set in the serial protocol / Geber 3: Fehlerbit im seriellen Protokoll gesetzt'; 33414 'Encoder 3: Amplitude error track C or D (C^2 + D^2) / Geber 3: Amplitudenfehler Spur C oder D (C^2 + D^2)'; 33415 'Encoder 3: Amplitude alarm track A or B (A^2 + B^2) / Geber 3: Amplitudenwarnung Spur A oder B (A^2 + B^2)'; 33418 'Encoder 3: Speed difference per sampling rate exceeded / Geber 3: Drehzahldifferenz je Abtastrate überschritten'; 33419 'Encoder 3: Track A or B outside tolerance / Geber 3: Spur A oder B außerhalb Toleranz'; 33421 'Encoder 3: Coarse position error / Geber 3: Groblage fehlerhaft'; 33422 'Encoder 3: Pulses per revolution square-wave encoder outside tolerance bandwidth Geber 3: Impulszahl Rechteckgeber außerhalb Toleranzband'; 33429 'Encoder 3: Position difference, hall sensor/track C/D and A/B too large Geber 3: Lagedifferenz Hallsensor/Spur C/D und Spur A/B zu groß'; 33431 'Encoder 3: Deviation, position incremental/absolute too large / Geber 3: Abweichung Lage inkrementell/absolut zu groß'; 33432 'Encoder 3: Rotor position adaptation corrects deviation / Geber 3: Rotorlageadaption korrigiert Abweichung'; 33442 'Encoder 3: Battery voltage pre-alarm / Geber 3: Batteriespannung Vorwarnung'; 33443 'Encoder 3: Unipolar CD signal level outside specification / Geber 3: Unipolar CD Signalpegel außerhalb Spezifikation'; 33460 'Encoder 3: Analog sensor channel A failed / Geber 3: Analogsensor Kanal A ausgefallen'; 33461 'Encoder 3: Analog sensor channel B failed / Geber 3: Analogsensor Kanal B ausgefallen'; 33462 'Encoder 3: Analog sensor, no channel active / Geber 3: Analogsensor Kein Kanal aktiv'; 33463 'Encoder 3: Analog sensor position value exceeds limit value / Geber 3: Analogsensor Lagewert überschreitet Grenzwert'; 33470 'Encoder 3: Soiling detected / Geber 3: Verschmutzung erkannt'; 33500 'Encoder 3: Position tracking traversing range exceeded / Geber 3: Lageverfolgung Verfahrbereich überschritten'; 33501 'Encoder 3: Position tracking encoder position outside tolerance window Geber 3: Lageverfolgung Geberposition außerhalb Toleranzfenster'; 33502 'Encoder 3: Encoder with measuring gear, without valid signals / Geber 3: Geber mit Messgetriebe ohne gültige Signale'; 33503 'Encoder 3: Position tracking cannot be reset / Geber 3: Lageverfolgung lässt sich nicht zurücksetzen'; 33700 'Encoder 3: Effectivity test does not supply the expected value / Geber 3: Wirksamkeitstest liefert nicht Erwartungswert'; 33800 'Encoder 3: Group signal / Geber 3: Sammelmeldung'; 33802 'Encoder 3: Time slice overflow / Geber 3: Zeitscheibenüberlauf'; 33804 'Encoder 3: Checksum error / Geber 3: Checksummenfehler'; 33805 'Encoder 3: EPROM checksum error / Geber 3: Prüfsumme EPROM nicht korrekt'; 33806 'Encoder 3: Initialization error / Geber 3: Initialisierung fehlgeschlagen'; 33811 'Encoder 3: Encoder serial number changed / Geber 3: Geberseriennummer geändert'; 33812 'Encoder 3: Requested cycle or RX-/TX timing not supported Geber 3: Angeforderter Zyklus bzw. RX-/TX-Timing nicht unterstützt'; 33813 'Encoder 3: Hardware logic unit failed / Geber 3: Hardware Logikeinheit ausgefallen'; 33850 'Encoder 3: Encoder evaluation, internal software error / Geber 3: Geberauswertung Softwarefehler intern'; 33898 'Encoder 3: POWER ON signal / Geber 3: POWER ON Meldung'; 33899 'Encoder 3: Unknown fault / Geber 3: Unbekannte Störung'; 33902 'Encoder 3: SPI-BUS error occurred / Geber 3: SPI-BUS Fehler aufgetreten'; 33903 'Encoder 3: I2C-BUS error occurred / Geber 3: I2C-BUS Fehler aufgetreten'; 33905 'Encoder 3: Parameterization error / Geber 3: Fehlparametrierung'; 33915 'Encoder 3: Configuration error / Geber 3: Konfigurationsfehler'; 33916 'Encoder 3: Parameterization fault / Geber 3: Fehler bei Parametrierung'; 33920 'Encoder 3: Temperature sensor fault / Geber 3: Fehler Temperatursensor'; 33930 'Encoder 3: Data logger has saved data / Geber 3: Datalogger hat Daten gespeichert'; 33940 'Sensor 3: Spindle clamping state error / Geber 3: Spindel Spannzustand fehlerhaft'; 33999 'Encoder 3: Unknown alarm / Geber 3: Unbekannte Warnung'; 35000 'TM54F: Sampling time invalid / TM54F: Abtastzeit ungültig'; 35001 'TM54F: Parameter value invalid / TM54F: Parameterwert ungültig'; 35002 'TM54F: Commissioning not possible / TM54F: Inbetriebnahmemodus nicht möglich'; 35003 'TM54F: Acknowledgement on the Control Unit is required / TM54F: Quittierung auf Control Unit erforderlich'; 35011 'TM54F: Drive object number assignment illegal / TM54F: Antriebsobjektnummer Zuordnung unzulässig'; 35012 'TM54F: Test stop active / TM54F: Teststop aktiv'; 35013 'TM54F: Test stop error / TM54F: Teststop fehlerhaft'; 35014 'TM54F: Test stop required / TM54F: Teststop notwendig'; 35015 'TM54F: Motor Module replaced or configuration inconsistent TM54F: Motor Module getauscht oder Konfiguration inkonsistent'; 35016 'TM54F: Net data communication with drive not established / TM54F: Nutzdatenkommunikation mit Antrieb nicht aufgebaut'; 35040 'TM54F: 24 V undervoltage / TM54F: Unterspannung 24 V'; 35043 'TM54F: 24 V overvoltage / TM54F: Überspannung 24 V'; 35051 'TM54F: Defect in a monitoring channel / TM54F: Defekt in einem Überwachungskanal'; 35052 'TM54F: Internal hardware error / TM54F: Hardwarefehler intern'; 35053 'TM54F: Temperature fault threshold exceeded / TM54F: Temperatur Störschwelle überschritten'; 35054 'TM54F: Temperature alarm threshold exceeded / TM54F: Temperatur Warnschwelle überschritten'; 35075 'TM54F: Error during internal communication / TM54F: Fehler bei interner Kommunikation'; 35080 'TM54F: Checksum error safety parameters / TM54F: Prüfsummenfehler sichere Parameter'; 35081 'TM54F: Static (steady state) 1 signal at the F-DI for safety-relevant acknowledgement TM54F: Statisches 1-Signal am F-DI für sichere Quittierung'; 35150 'TM54F: Communication error / TM54F: Kommunikationsfehler'; 35151 'TM54F: Discrepancy error / TM54F: Diskrepanzfehler'; 35152 'TM54F: Internal software error / TM54F: Softwarefehler intern'; 35200 'TM: Calibration data / TM: Kalibrierdaten'; 35207 'TM: Temperature fault/alarm threshold channel 1 exceeded / TM: Temperatur Stör-/Warnschwelle Kanal 1 überschritten'; 35208 'TM: Temperature fault/alarm threshold channel 2 exceeded / TM: Temperatur Stör-/Warnschwelle Kanal 2 überschritten'; 35209 'TM: Temperature fault/alarm threshold channel 3 exceeded / TM: Temperatur Stör-/Warnschwelle Kanal 3 überschritten'; 35210 'TM: Temperature fault/alarm threshold channel 4 exceeded / TM: Temperatur Stör-/Warnschwelle Kanal 4 überschritten'; 35211 'TM: Temperature alarm threshold channel 1 exceeded / TM: Temperatur Warnschwelle Kanal 1 überschritten'; 35212 'TM: Temperature alarm threshold channel 2 exceeded / TM: Temperatur Warnschwelle Kanal 2 überschritten'; 35213 'TM: Temperature alarm threshold channel 3 exceeded / TM: Temperatur Warnschwelle Kanal 3 überschritten'; 35214 'TM: Temperature alarm threshold channel 4 exceeded / TM: Temperatur Warnschwelle Kanal 4 überschritten'; 35220 'TM: Frequency limit reached for signal output / TM: Grenzfrequenz für Signalausgabe erreicht'; 35221 'TM: Setpoint - actual value deviation, outside the tolerance range TM: Soll-Ist-Abweichung außerhalb Toleranz'; 35222 'TM: Encoder pulse number not permissible / TM: Geberstrichzahl unzulässig'; 35223 'TM: Zero mark offset not permissible / TM: Nullmarkenoffset unzulässig'; 35224 'TM: Zero mark synchronization interrupted / TM: Nullmarkensynchronisation abgebrochen'; 35225 'TM: Zero mark synchronization held - encoder not in the ready state TM: Nullmarkensynchronisation angehalten - Geber nicht im Zustand bereit'; 35226 'TM: Tracks A/B are de-activated / TM: Spuren A/B sind deaktiviert'; 35227 'EDS changeover/encoder data set change not supported / EDS-Umschaltung/Geberdatensatz-à„nderung nicht unterstützt'; 35228 'TM: Sampling time p4099[3] invalid / TM: Abtastzeit p4099[3] ungültig'; 35229 'TM: Time slice de-activated / TM: Zeitscheibe deaktiviert'; 35230 'TM: Hardware fault / TM: Hardware fehlerhaft'; 35231 'TM: Master control by PLC missing / TM: Führung durch PLC fehlt'; 35232 'TM41: Zero mark no longer synchronous POWER ON required / TM41: Nullmarke nicht mehr synchron POWER ON erforderlich'; 35800 'TM: Group signal / TM: Sammelmeldung'; 35802 'TM: Time slice overflow / TM: Zeitscheibenüberlauf'; 35803 'TM: Memory test / TM: Speichertest'; 35804 'TM: CRC'; 35805 'TM: EPROM checksum error / TM: Prüfsumme EPROM nicht korrekt'; 35807 'TM: Sequence control time monitoring / TM: Ablaufsteuerung Zeitüberwachung'; 35850 'TM: Internal software error / TM: Softwarefehler intern'; 35898 'TM: POWER ON signal / TM: POWER ON Meldung'; 35899 'TM: Unknown fault / TM: Unbekannte Störung'; 35903 'TM: I2C bus error occurred / TM: I2C-Bus Fehler aufgetreten'; 35904 'TM: EEPROM'; 35905 'TM: Parameter access / TM: Parameterzugriff'; 35906 'TM: 24 V power supply missing / TM: Spannungsversorgung 24 V fehlt'; 35907 'TM: Hardware initialization error / TM: Initialisierung Hardware fehlgeschlagen'; 35910 'TM: Module overtemperature / TM: Übertemperatur im Modul'; 35911 'TM: Clock synchronous operation sign-of-life missing / TM: Taktsynchroner Betrieb Lebenszeichenausfall'; 35920 'TM: Error temperature sensor channel 1 / TM: Fehler Temperatursensor Kanal 1'; 35921 'TM: Error temperature sensor channel 2 / TM: Fehler Temperatursensor Kanal 2'; 35922 'TM: Error temperature sensor channel 3 / TM: Fehler Temperatursensor Kanal 3'; 35923 'TM: Error temperature sensor channel 4 / TM: Fehler Temperatursensor Kanal 4'; 35999 'TM: Unknown alarm / TM: Unbekannte Warnung'; 36207 'Hub: Overtemperature component / Hub: Übertemperaturfehler Komponente'; 36211 'Hub: Overtemperature alarm component / Hub: Übertemperaturwarnung Komponente'; 36214 'Hub: overvoltage fault 24 V supply / Hub: Überspannungsfehler 24-V-Versorgung'; 36216 'Hub: undervoltage fault 24 V supply / Hub: Unterspannungsfehler 24-V-Versorgung'; 36217 'Hub: undervoltage alarm 24 V supply / Hub Unterspannungswarnung 24-V-Versorgung'; 36800 'Hub: Group signal / Hub: Sammelmeldung'; 36802 'Hub: Time slice overflow / Hub: Zeitscheibenüberlauf'; 36804 'Hub: Checksum error / Hub: Checksummenfehler'; 36805 'Hub: EEPROM checksum incorrect / Hub: EEPROM Prüfsumme nicht korrekt'; 36898 'Hub: POWER ON signal / Hub: POWER ON Meldung'; 36899 'Hub: Unknown fault / Hub: Unbekannte Störung'; 36999 'Hub: Unknown alarm / Hub: Unbekannte Warnung'; 37001 'HF damping module: Overcurrent / HF-Dämpfungsmodul: Überstrom'; 37002 'HF damping module: Damping voltage too high / HF-Dämpfungsmodul: Dämpfungsspannung zu hoch'; 37004 'HF damping module: Heat sink overtemperature / HF-Dämpfungsmodul: Übertemperatur Kühlkörper'; 37005 'HF damping module: I2t overload / HF-Dämpfungsmodul: Überlastung I2t'; 37012 'HF damping module: Temperature sensor heat sink wire breakage HF-Dämpfungsmodul: Temperaturfühler Kühlkörper Drahtbruch'; 37013 'HF damping module: Temperature sensor heat sink short circuit / HF-Dämpfungsmodul: Temperaturfühler Kühlkörper Kurzschluss'; 37024 'HF damping module: Overtemperature thermal model / HF-Dämpfungsmodul: Übertemperatur Thermisches Modell'; 37025 'HF damping module: Overtemperature chip / HF-Dämpfungsmodul: Übertemperatur Chip'; 37034 'HF damping module: Internal overtemperature / HF-Dämpfungsmodul: Übertemperatur Innenraum'; 37036 'HF 